C05414=1035.741,-69.357,-80.600,168.332,38.927,157.287
C05415=1035.746,-69.108,-80.612,168.335,38.926,157.287
C05416=1035.752,-68.858,-80.623,168.337,38.926,157.287
C05417=1035.758,-68.609,-80.635,168.340,38.926,157.287
C05418=1035.766,-68.326,-80.648,168.343,38.925,157.287
C05419=1035.773,-68.043,-80.661,168.346,38.925,157.287
C05420=1035.779,-67.760,-80.674,168.349,38.924,157.287
C05421=1035.786,-67.478,-80.687,168.352,38.924,157.287
C05422=1035.793,-67.228,-80.699,168.354,38.923,157.287
C05423=1035.798,-66.978,-80.711,168.357,38.923,157.287
C05424=1035.804,-66.729,-80.723,168.359,38.922,157.287
C05425=1035.811,-66.479,-80.735,168.362,38.922,157.287
C05426=1035.817,-66.229,-80.746,168.365,38.921,157.287
C05427=1035.823,-65.980,-80.758,168.367,38.921,157.287
C05428=1035.829,-65.730,-80.769,168.370,38.921,157.287
C05429=1035.836,-65.480,-80.781,168.371,38.920,157.287
C05430=1035.842,-65.231,-80.793,168.374,38.920,157.287
C05431=1035.847,-64.981,-80.805,168.376,38.919,157.287
C05432=1035.854,-64.731,-80.817,168.379,38.919,157.287
C05433=1035.860,-64.482,-80.828,168.382,38.918,157.287
C05434=1035.866,-64.232,-80.840,168.384,38.918,157.287
C05435=1035.872,-63.982,-80.852,168.387,38.918,157.287
C05436=1035.878,-63.733,-80.864,168.389,38.917,157.287
C05437=1035.885,-63.483,-80.875,168.392,38.917,157.287
C05438=1035.891,-63.234,-80.887,168.394,38.916,157.287
C05439=1035.897,-62.984,-80.899,168.397,38.916,157.287
C05440=1035.903,-62.734,-80.910,168.400,38.915,157.287
C05441=1035.910,-62.485,-80.922,168.402,38.915,157.287
C05442=1035.916,-62.235,-80.934,168.405,38.914,157.287
C05443=1035.921,-61.986,-80.946,168.407,38.914,157.287
C05444=1035.928,-61.736,-80.958,168.410,38.914,157.287
C05445=1035.934,-61.486,-80.970,168.412,38.913,157.287
C05446=1035.940,-61.236,-80.982,168.415,38.913,157.287
C05447=1035.946,-60.987,-80.994,168.418,38.912,157.287
C05448=1035.953,-60.737,-81.005,168.420,38.912,157.287
C05449=1035.959,-60.488,-81.017,168.423,38.911,157.287
C05450=1035.965,-60.238,-81.030,168.425,38.911,157.287
C05451=1035.972,-59.988,-81.042,168.428,38.910,157.287
C05452=1035.978,-59.739,-81.053,168.430,38.910,157.287
C05453=1035.984,-59.489,-81.066,168.433,38.909,157.287
C05454=1035.990,-59.239,-81.077,168.435,38.909,157.287
C05455=1035.997,-58.990,-81.089,168.438,38.908,157.287
C05456=1036.004,-58.740,-81.101,168.441,38.908,157.287
C05457=1036.009,-58.491,-81.113,168.443,38.908,157.287
C05458=1036.015,-58.241,-81.125,168.446,38.907,157.287
C05459=1036.022,-57.992,-81.137,168.448,38.907,157.287
C05460=1036.028,-57.742,-81.150,168.451,38.906,157.287
C05461=1036.034,-57.492,-81.161,168.453,38.906,157.287
C05462=1036.041,-57.242,-81.173,168.456,38.906,157.287
C05463=1036.046,-56.993,-81.185,168.458,38.905,157.287
C05464=1036.053,-56.743,-81.197,168.461,38.905,157.287
C05465=1036.060,-56.494,-81.209,168.464,38.904,157.287
C05466=1036.066,-56.248,-81.221,168.466,38.904,157.287
C05467=1036.072,-56.003,-81.233,168.469,38.904,157.287
C05468=1036.078,-55.758,-81.245,168.470,38.903,157.287
C05469=1036.084,-55.512,-81.257,168.473,38.903,157.287
C05470=1036.090,-55.268,-81.269,168.475,38.902,157.286
C05471=1036.097,-55.022,-81.280,168.478,38.902,157.287
C05472=1036.103,-54.777,-81.293,168.480,38.902,157.287
C05473=1036.109,-54.531,-81.304,168.483,38.901,157.286
C05474=1036.115,-54.282,-81.316,168.485,38.901,157.287
C05475=1036.122,-54.032,-81.328,168.488,38.901,157.287
C05476=1036.128,-53.782,-81.341,168.490,38.900,157.286
C05477=1036.135,-53.533,-81.353,168.493,38.900,157.287
C05478=1036.141,-53.283,-81.365,168.495,38.899,157.286
C05479=1036.147,-53.033,-81.377,168.498,38.899,157.286
C05480=1036.154,-52.784,-81.389,168.500,38.899,157.287
C05481=1036.160,-52.534,-81.401,168.503,38.898,157.286
C05482=1036.168,-52.244,-81.416,168.506,38.898,157.286
C05483=1036.174,-51.954,-81.430,168.509,38.897,157.286
C05484=1036.182,-51.664,-81.444,168.512,38.897,157.286
C05485=1036.190,-51.373,-81.459,168.515,38.896,157.286
C05486=1036.197,-51.124,-81.471,168.517,38.896,157.286
C05487=1036.203,-50.874,-81.483,168.520,38.895,157.286
C05488=1036.209,-50.624,-81.495,168.522,38.895,157.286
C05489=1036.216,-50.375,-81.507,168.525,38.894,157.286
C05490=1036.222,-50.125,-81.520,168.527,38.894,157.286
C05491=1036.228,-49.876,-81.533,168.530,38.894,157.287
C05492=1036.234,-49.626,-81.546,168.532,38.894,157.287
C05493=1036.240,-49.377,-81.557,168.535,38.894,157.287
C05494=1036.246,-49.127,-81.570,168.537,38.893,157.287
C05495=1036.252,-48.878,-81.583,168.539,38.893,157.287
C05496=1036.259,-48.628,-81.595,168.542,38.893,157.287
C05497=1036.265,-48.378,-81.607,168.544,38.893,157.287
C05498=1036.270,-48.129,-81.620,168.547,38.892,157.287
C05499=1036.277,-47.880,-81.633,168.549,38.892,157.287
C05500=1036.283,-47.630,-81.645,168.552,38.892,157.287
C05501=1036.289,-47.380,-81.658,168.554,38.892,157.287
C05502=1036.295,-47.131,-81.671,168.557,38.891,157.287
C05503=1036.302,-46.881,-81.683,168.559,38.891,157.287
C05504=1036.308,-46.631,-81.696,168.562,38.891,157.287
C05505=1036.314,-46.382,-81.709,168.564,38.891,157.287
C05506=1036.320,-46.132,-81.721,168.566,38.891,157.287
C05507=1036.327,-45.882,-81.733,168.569,38.890,157.287
C05508=1036.333,-45.633,-81.747,168.571,38.890,157.287
C05509=1036.339,-45.383,-81.759,168.574,38.889,157.287
C05510=1036.345,-45.134,-81.771,168.576,38.889,157.287
C05511=1036.352,-44.884,-81.785,168.579,38.889,157.287
C05512=1036.358,-44.634,-81.797,168.581,38.889,157.287
C05513=1036.364,-44.385,-81.811,168.584,38.889,157.287
C05514=1036.371,-44.135,-81.823,168.586,38.889,157.287
C05515=1036.377,-43.885,-81.835,168.588,38.889,157.287
C05516=1036.383,-43.636,-81.848,168.591,38.888,157.287
C05517=1036.389,-43.386,-81.861,168.593,38.888,157.287
C05518=1036.396,-43.137,-81.874,168.596,38.887,157.287
C05519=1036.402,-42.887,-81.886,168.598,38.887,157.287
C05520=1036.408,-42.638,-81.899,168.601,38.887,157.287
C05521=1036.414,-42.388,-81.912,168.603,38.887,157.287
C05522=1036.421,-42.139,-81.925,168.606,38.887,157.287
C05523=1036.428,-41.888,-81.938,168.608,38.887,157.287
C05524=1036.434,-41.639,-81.951,168.610,38.887,157.287
C05525=1036.440,-41.389,-81.963,168.613,38.886,157.287
C05526=1036.446,-41.140,-81.977,168.615,38.886,157.287
C05527=1036.453,-40.890,-81.989,168.618,38.885,157.287
C05528=1036.459,-40.641,-82.002,168.620,38.885,157.287
C05529=1036.465,-40.391,-82.014,168.623,38.885,157.287
C05530=1036.471,-40.141,-82.028,168.625,38.885,157.287
C05531=1036.478,-39.892,-82.040,168.627,38.885,157.287
C05532=1036.484,-39.642,-82.053,168.630,38.885,157.288
C05533=1036.490,-39.393,-82.066,168.632,38.885,157.288
C05534=1036.496,-39.143,-82.079,168.635,38.884,157.287
C05535=1036.502,-38.893,-82.092,168.637,38.884,157.288
C05536=1036.510,-38.644,-82.105,168.640,38.883,157.288
C05537=1036.515,-38.394,-82.119,168.642,38.883,157.288
C05538=1036.521,-38.144,-82.131,168.644,38.883,157.288
C05539=1036.528,-37.895,-82.144,168.647,38.883,157.288
C05540=1036.534,-37.646,-82.158,168.649,38.883,157.288
C05541=1036.540,-37.396,-82.170,168.651,38.883,157.288
C05542=1036.546,-37.146,-82.184,168.654,38.883,157.288
C05543=1036.553,-36.897,-82.197,168.656,38.883,157.288
C05544=1036.559,-36.647,-82.210,168.659,38.883,157.288
C05545=1036.565,-36.398,-82.223,168.662,38.883,157.288
C05546=1036.572,-36.117,-82.238,168.665,38.883,157.288
C05547=1036.580,-35.835,-82.253,168.667,38.882,157.288
C05548=1036.586,-35.554,-82.267,168.670,38.882,157.288
C05549=1036.593,-35.273,-82.282,168.673,38.882,157.288
C05550=1036.600,-35.024,-82.296,168.675,38.882,157.288
C05551=1036.606,-34.774,-82.308,168.677,38.882,157.288
C05552=1036.612,-34.524,-82.322,168.680,38.882,157.288
C05553=1036.619,-34.275,-82.335,168.682,38.882,157.288
C05554=1036.625,-34.026,-82.348,168.684,38.881,157.288
C05555=1036.631,-33.776,-82.361,168.687,38.881,157.288
C05556=1036.638,-33.526,-82.375,168.689,38.881,157.288
C05557=1036.644,-33.277,-82.388,168.692,38.881,157.289
C05558=1036.650,-33.027,-82.401,168.694,38.881,157.289
C05559=1036.655,-32.778,-82.415,168.696,38.881,157.289
C05560=1036.662,-32.528,-82.429,168.699,38.880,157.289
C05561=1036.668,-32.278,-82.441,168.701,38.880,157.289
C05562=1036.674,-32.029,-82.454,168.703,38.880,157.289
C05563=1036.681,-31.780,-82.468,168.706,38.880,157.289
C05564=1036.687,-31.530,-82.481,168.708,38.880,157.289
C05565=1036.694,-31.280,-82.495,168.710,38.880,157.289
C05566=1036.700,-31.031,-82.508,168.713,38.880,157.289
C05567=1036.707,-30.781,-82.521,168.715,38.880,157.289
C05568=1036.713,-30.532,-82.535,168.717,38.880,157.289
C05569=1036.719,-30.283,-82.548,168.720,38.880,157.289
C05570=1036.726,-30.032,-82.561,168.722,38.880,157.289
C05571=1036.732,-29.783,-82.574,168.725,38.880,157.289
C05572=1036.738,-29.533,-82.587,168.727,38.879,157.289
C05573=1036.745,-29.283,-82.601,168.729,38.879,157.289
C05574=1036.751,-29.034,-82.614,168.732,38.879,157.289
C05575=1036.757,-28.785,-82.628,168.734,38.879,157.289
C05576=1036.763,-28.535,-82.642,168.736,38.879,157.289
C05577=1036.770,-28.285,-82.655,168.739,38.879,157.289
C05578=1036.776,-28.036,-82.668,168.741,38.879,157.289
C05579=1036.783,-27.786,-82.682,168.743,38.878,157.289
C05580=1036.789,-27.537,-82.695,168.746,38.878,157.289
C05581=1036.796,-27.287,-82.709,168.748,38.878,157.290
C05582=1036.802,-27.038,-82.722,168.750,38.878,157.290
C05583=1036.807,-26.788,-82.736,168.753,38.878,157.290
C05584=1036.814,-26.538,-82.750,168.755,38.878,157.290
C05585=1036.820,-26.289,-82.763,168.757,38.878,157.290
C05586=1036.826,-26.039,-82.777,168.761,38.878,157.290
C05587=1036.833,-25.789,-82.791,168.763,38.878,157.290
C05588=1036.839,-25.541,-82.804,168.765,38.878,157.290
C05589=1036.846,-25.291,-82.818,168.767,38.878,157.290
C05590=1036.851,-25.041,-82.832,168.770,38.878,157.290
C05591=1036.858,-24.792,-82.845,168.772,38.878,157.290
C05592=1036.865,-24.542,-82.859,168.774,38.878,157.290
C05593=1036.870,-24.292,-82.873,168.777,38.878,157.290
C05594=1036.876,-24.043,-82.886,168.779,38.878,157.290
C05595=1036.883,-23.793,-82.901,168.781,38.878,157.290
C05596=1036.889,-23.544,-82.914,168.783,38.878,157.290
C05597=1036.896,-23.294,-82.928,168.786,38.878,157.290
C05598=1036.901,-23.045,-82.942,168.788,38.878,157.290
C05599=1036.908,-22.795,-82.955,168.790,38.878,157.291
C05600=1036.914,-22.546,-82.969,168.793,38.878,157.291
C05601=1036.920,-22.296,-82.983,168.795,38.878,157.291
C05602=1036.927,-22.046,-82.997,168.797,38.878,157.291
C05603=1036.933,-21.797,-83.010,168.799,38.878,157.291
C05604=1036.939,-21.548,-83.025,168.802,38.877,157.291
C05605=1036.946,-21.298,-83.038,168.804,38.878,157.291
C05606=1036.952,-21.048,-83.052,168.806,38.878,157.291
C05607=1036.958,-20.799,-83.066,168.809,38.878,157.291
C05608=1036.965,-20.549,-83.080,168.811,38.878,157.291
C05609=1036.971,-20.300,-83.093,168.813,38.877,157.291
C05610=1036.979,-20.018,-83.110,168.817,38.878,157.291
C05611=1036.985,-19.736,-83.125,168.819,38.878,157.291
C05612=1036.992,-19.454,-83.141,168.822,38.878,157.291
C05613=1036.999,-19.172,-83.157,168.824,38.877,157.291
C05614=1037.006,-18.923,-83.171,168.827,38.877,157.291
C05615=1037.013,-18.673,-83.184,168.829,38.878,157.292
C05616=1037.018,-18.424,-83.198,168.831,38.878,157.292
C05617=1037.025,-18.174,-83.213,168.833,38.878,157.292
C05618=1037.031,-17.925,-83.226,168.836,38.877,157.292
C05619=1037.038,-17.675,-83.240,168.838,38.877,157.292
C05620=1037.044,-17.426,-83.254,168.840,38.877,157.292
C05621=1037.050,-17.176,-83.268,168.843,38.878,157.292
C05622=1037.056,-16.927,-83.282,168.845,38.877,157.292
C05623=1037.063,-16.677,-83.296,168.847,38.877,157.292
C05624=1037.070,-16.427,-83.310,168.849,38.877,157.292
C05625=1037.076,-16.178,-83.324,168.852,38.877,157.292
C05626=1037.082,-15.928,-83.338,168.854,38.878,157.292
C05627=1037.089,-15.680,-83.352,168.856,38.877,157.292
C05628=1037.095,-15.430,-83.366,168.858,38.877,157.292
C05629=1037.101,-15.180,-83.380,168.861,38.877,157.292
C05630=1037.107,-14.930,-83.395,168.863,38.878,157.292
C05631=1037.114,-14.681,-83.408,168.865,38.877,157.293
C05632=1037.120,-14.431,-83.423,168.867,38.877,157.293
C05633=1037.127,-14.182,-83.437,168.870,38.878,157.293
C05634=1037.133,-13.933,-83.451,168.873,38.878,157.293
C05635=1037.139,-13.683,-83.466,168.875,38.878,157.293
C05636=1037.145,-13.434,-83.479,168.877,38.878,157.293
C05637=1037.152,-13.184,-83.494,168.879,38.878,157.293
C05638=1037.157,-12.934,-83.508,168.882,38.878,157.293
C05639=1037.164,-12.685,-83.523,168.884,38.878,157.293
C05640=1037.170,-12.435,-83.537,168.886,38.878,157.293
C05641=1037.176,-12.186,-83.551,168.888,38.878,157.293
C05642=1037.183,-11.936,-83.566,168.890,38.879,157.293
C05643=1037.189,-11.687,-83.580,168.893,38.878,157.293
C05644=1037.196,-11.438,-83.594,168.895,38.878,157.293
C05645=1037.202,-11.188,-83.609,168.897,38.878,157.293
C05646=1037.208,-10.938,-83.623,168.899,38.879,157.294
C05647=1037.215,-10.689,-83.637,168.901,38.879,157.294
C05648=1037.221,-10.439,-83.651,168.904,38.878,157.294
C05649=1037.227,-10.190,-83.666,168.906,38.879,157.294
C05650=1037.234,-9.940,-83.680,168.908,38.879,157.294
C05651=1037.239,-9.691,-83.694,168.910,38.879,157.294
C05652=1037.246,-9.441,-83.709,168.913,38.879,157.294
C05653=1037.253,-9.192,-83.723,168.916,38.879,157.294
C05654=1037.258,-8.943,-83.738,168.918,38.879,157.294
C05655=1037.264,-8.693,-83.752,168.920,38.879,157.294
C05656=1037.272,-8.443,-83.767,168.922,38.879,157.294
C05657=1037.277,-8.194,-83.781,168.924,38.879,157.294
C05658=1037.283,-7.944,-83.795,168.927,38.880,157.295
C05659=1037.291,-7.695,-83.810,168.929,38.880,157.295
C05660=1037.297,-7.445,-83.825,168.931,38.879,157.295
C05661=1037.303,-7.196,-83.839,168.933,38.880,157.295
C05662=1037.310,-6.946,-83.853,168.935,38.880,157.295
C05663=1037.316,-6.696,-83.868,168.938,38.880,157.295
C05664=1037.322,-6.447,-83.882,168.940,38.880,157.295
C05665=1037.328,-6.198,-83.897,168.942,38.880,157.295
C05666=1037.335,-5.948,-83.911,168.944,38.880,157.295
C05667=1037.341,-5.698,-83.926,168.946,38.880,157.295
C05668=1037.347,-5.449,-83.941,168.949,38.880,157.295
C05669=1037.354,-5.200,-83.955,168.951,38.880,157.295
C05670=1037.361,-4.950,-83.970,168.953,38.880,157.295
C05671=1037.367,-4.701,-83.985,168.956,38.881,157.295
C05672=1037.373,-4.451,-83.998,168.958,38.880,157.296
C05673=1037.380,-4.202,-84.013,168.960,38.880,157.296
C05674=1037.387,-3.918,-84.029,168.963,38.881,157.296
C05675=1037.394,-3.635,-84.046,168.965,38.881,157.296
C05676=1037.402,-3.351,-84.063,168.968,38.881,157.296
C05677=1037.408,-3.067,-84.080,168.970,38.881,157.296
C05678=1037.414,-2.818,-84.095,168.972,38.881,157.296
C05679=1037.420,-2.569,-84.110,168.975,38.881,157.296
C05680=1037.427,-2.319,-84.125,168.977,38.882,157.296
C05681=1037.433,-2.069,-84.139,168.979,38.882,157.296
C05682=1037.439,-1.820,-84.154,168.981,38.882,157.296
C05683=1037.445,-1.571,-84.169,168.983,38.882,157.297
C05684=1037.452,-1.321,-84.184,168.985,38.883,157.297
C05685=1037.458,-1.071,-84.199,168.987,38.882,157.297
C05686=1037.464,-0.823,-84.213,168.990,38.883,157.297
C05687=1037.470,-0.573,-84.228,168.993,38.883,157.297
C05688=1037.476,-0.323,-84.243,168.995,38.883,157.297
C05689=1037.483,-0.074,-84.258,168.997,38.883,157.297
C05690=1037.489,0.175,-84.273,168.999,38.884,157.297
C05691=1037.495,0.425,-84.288,169.001,38.884,157.297
C05692=1037.501,0.675,-84.303,169.003,38.884,157.297
C05693=1037.508,0.924,-84.318,169.005,38.884,157.297
C05694=1037.514,1.173,-84.333,169.007,38.885,157.298
C05695=1037.520,1.422,-84.348,169.009,38.884,157.298
C05696=1037.527,1.672,-84.363,169.012,38.884,157.298
C05697=1037.533,1.922,-84.378,169.014,38.885,157.298
C05698=1037.539,2.171,-84.393,169.016,38.885,157.298
C05699=1037.546,2.421,-84.408,169.019,38.885,157.298
C05700=1037.552,2.671,-84.423,169.021,38.885,157.298
C05701=1037.558,2.920,-84.437,169.023,38.886,157.298
C05702=1037.565,3.169,-84.453,169.025,38.885,157.298
C05703=1037.571,3.418,-84.468,169.027,38.886,157.298
C05704=1037.577,3.668,-84.483,169.029,38.886,157.298
C05705=1037.584,3.918,-84.498,169.032,38.886,157.299
C05706=1037.590,4.167,-84.513,169.034,38.886,157.299
C05707=1037.595,4.417,-84.528,169.036,38.887,157.299
C05708=1037.602,4.666,-84.544,169.038,38.887,157.299
C05709=1037.608,4.915,-84.559,169.040,38.887,157.299
C05710=1037.615,5.165,-84.573,169.042,38.887,157.299
C05711=1037.621,5.415,-84.588,169.044,38.888,157.299
C05712=1037.627,5.664,-84.603,169.046,38.887,157.299
C05713=1037.634,5.913,-84.619,169.049,38.888,157.299
C05714=1037.641,6.163,-84.634,169.052,38.888,157.299
C05715=1037.647,6.413,-84.649,169.054,38.888,157.299
C05716=1037.653,6.662,-84.663,169.056,38.888,157.300
C05717=1037.659,6.911,-84.679,169.058,38.888,157.300
C05718=1037.666,7.160,-84.694,169.060,38.889,157.300
C05719=1037.672,7.410,-84.709,169.062,38.888,157.300
C05720=1037.679,7.660,-84.724,169.064,38.889,157.300
C05721=1037.685,7.909,-84.740,169.066,38.889,157.300
C05722=1037.691,8.159,-84.755,169.068,38.889,157.300
C05723=1037.697,8.408,-84.770,169.070,38.889,157.300
C05724=1037.704,8.657,-84.786,169.073,38.890,157.300
C05725=1037.710,8.907,-84.801,169.075,38.890,157.300
C05726=1037.717,9.157,-84.816,169.077,38.889,157.300
C05727=1037.723,9.406,-84.831,169.080,38.890,157.301
C05728=1037.730,9.655,-84.846,169.082,38.890,157.301
C05729=1037.736,9.905,-84.861,169.084,38.890,157.301
C05730=1037.743,10.154,-84.877,169.086,38.890,157.301
C05731=1037.749,10.404,-84.892,169.088,38.891,157.301
C05732=1037.756,10.653,-84.907,169.090,38.891,157.301
C05733=1037.762,10.902,-84.922,169.092,38.891,157.301
C05734=1037.768,11.152,-84.938,169.095,38.891,157.301
C05735=1037.774,11.402,-84.953,169.097,38.891,157.301
C05736=1037.781,11.651,-84.969,169.099,38.891,157.301
C05737=1037.787,11.901,-84.984,169.101,38.891,157.301
C05738=1037.795,12.186,-85.001,169.103,38.892,157.301
C05739=1037.802,12.471,-85.019,169.106,38.892,157.302
C05740=1037.810,12.757,-85.036,169.108,38.892,157.302
C05741=1037.817,13.042,-85.054,169.110,38.892,157.302
C05742=1037.824,13.291,-85.069,169.114,38.892,157.302
C05743=1037.830,13.541,-85.084,169.116,38.892,157.302
C05744=1037.836,13.790,-85.100,169.118,38.893,157.302
C05745=1037.843,14.040,-85.115,169.120,38.893,157.302
C05746=1037.849,14.289,-85.131,169.122,38.893,157.302
C05747=1037.856,14.538,-85.146,169.124,38.893,157.302
C05748=1037.862,14.788,-85.162,169.126,38.894,157.302
C05749=1037.868,15.037,-85.177,169.128,38.893,157.302
C05750=1037.875,15.287,-85.193,169.130,38.894,157.303
C05751=1037.880,15.536,-85.208,169.132,38.895,157.303
C05752=1037.887,15.786,-85.224,169.134,38.894,157.303
C05753=1037.893,16.035,-85.240,169.136,38.895,157.303
C05754=1037.899,16.285,-85.255,169.138,38.895,157.303
C05755=1037.906,16.534,-85.271,169.141,38.895,157.303
C05756=1037.912,16.784,-85.286,169.143,38.895,157.303
C05757=1037.918,17.033,-85.302,169.145,38.896,157.303
C05758=1037.925,17.282,-85.318,169.147,38.896,157.303
C05759=1037.931,17.532,-85.333,169.149,38.896,157.304
C05760=1037.937,17.781,-85.349,169.151,38.897,157.304
C05761=1037.943,18.030,-85.365,169.153,38.896,157.304
C05762=1037.950,18.280,-85.381,169.156,38.897,157.304
C05763=1037.957,18.529,-85.396,169.158,38.897,157.304
C05764=1037.963,18.779,-85.412,169.160,38.897,157.304
C05765=1037.969,19.028,-85.427,169.162,38.897,157.304
C05766=1037.976,19.277,-85.443,169.164,38.898,157.304
C05767=1037.982,19.527,-85.459,169.167,38.898,157.304
C05768=1037.988,19.776,-85.474,169.169,38.898,157.304
C05769=1037.994,20.026,-85.491,169.171,38.899,157.305
C05770=1038.001,20.275,-85.506,169.173,38.899,157.305
C05771=1038.007,20.525,-85.522,169.175,38.899,157.305
C05772=1038.014,20.775,-85.538,169.177,38.900,157.305
C05773=1038.020,21.024,-85.554,169.179,38.899,157.305
C05774=1038.027,21.273,-85.570,169.181,38.900,157.305
C05775=1038.033,21.522,-85.586,169.183,38.900,157.305
C05776=1038.039,21.772,-85.601,169.185,38.900,157.305
C05777=1038.045,22.021,-85.617,169.187,38.901,157.305
C05778=1038.052,22.270,-85.633,169.189,38.901,157.305
C05779=1038.058,22.520,-85.649,169.192,38.901,157.306
C05780=1038.065,22.769,-85.665,169.194,38.902,157.306
C05781=1038.071,23.019,-85.681,169.196,38.902,157.306
C05782=1038.077,23.268,-85.696,169.198,38.902,157.306
C05783=1038.083,23.518,-85.713,169.200,38.902,157.306
C05784=1038.090,23.767,-85.728,169.202,38.903,157.306
C05785=1038.096,24.016,-85.744,169.204,38.903,157.306
C05786=1038.102,24.265,-85.761,169.206,38.903,157.306
C05787=1038.109,24.516,-85.776,169.208,38.904,157.306
C05788=1038.115,24.765,-85.792,169.210,38.903,157.307
C05789=1038.121,25.014,-85.808,169.212,38.904,157.307
C05790=1038.127,25.264,-85.824,169.215,38.904,157.307
C05791=1038.134,25.513,-85.840,169.217,38.904,157.307
C05792=1038.141,25.763,-85.856,169.219,38.905,157.307
C05793=1038.147,26.012,-85.872,169.221,38.905,157.307
C05794=1038.153,26.261,-85.888,169.223,38.905,157.307
C05795=1038.159,26.510,-85.905,169.225,38.906,157.307
C05796=1038.166,26.759,-85.920,169.227,38.906,157.307
C05797=1038.172,27.009,-85.937,169.229,38.906,157.308
C05798=1038.179,27.258,-85.953,169.231,38.906,157.308
C05799=1038.185,27.508,-85.969,169.233,38.907,157.308
C05800=1038.191,27.758,-85.984,169.235,38.907,157.308
C05801=1038.198,28.008,-86.000,169.237,38.907,157.308
C05802=1038.205,28.294,-86.019,169.240,38.907,157.308
C05803=1038.212,28.580,-86.038,169.243,38.908,157.308
C05804=1038.219,28.867,-86.056,169.245,38.908,157.308
C05805=1038.226,29.153,-86.075,169.247,38.908,157.308
C05806=1038.233,29.404,-86.092,169.249,38.909,157.309
C05807=1038.239,29.653,-86.108,169.251,38.909,157.309
C05808=1038.246,29.902,-86.123,169.253,38.910,157.309
C05809=1038.252,30.151,-86.140,169.255,38.910,157.309
C05810=1038.258,30.401,-86.156,169.257,38.910,157.309
C05811=1038.264,30.650,-86.173,169.260,38.911,157.309
C05812=1038.271,30.899,-86.189,169.262,38.911,157.309
C05813=1038.277,31.148,-86.205,169.264,38.911,157.309
C05814=1038.284,31.398,-86.222,169.266,38.912,157.310
C05815=1038.290,31.648,-86.238,169.268,38.912,157.310
C05816=1038.296,31.897,-86.254,169.270,38.912,157.310
C05817=1038.302,32.146,-86.270,169.272,38.913,157.310
C05818=1038.309,32.396,-86.287,169.274,38.912,157.310
C05819=1038.315,32.645,-86.304,169.276,38.913,157.310
C05820=1038.321,32.894,-86.320,169.278,38.913,157.310
C05821=1038.327,33.144,-86.336,169.280,38.913,157.310
C05822=1038.334,33.393,-86.352,169.283,38.914,157.310
C05823=1038.340,33.643,-86.368,169.285,38.914,157.311
C05824=1038.346,33.891,-86.385,169.287,38.915,157.311
C05825=1038.353,34.142,-86.402,169.289,38.915,157.311
C05826=1038.360,34.391,-86.418,169.291,38.915,157.311
C05827=1038.366,34.640,-86.434,169.293,38.916,157.311
C05828=1038.372,34.890,-86.451,169.295,38.916,157.311
C05829=1038.378,35.139,-86.467,169.297,38.916,157.311
C05830=1038.384,35.388,-86.484,169.299,38.917,157.311
C05831=1038.392,35.638,-86.500,169.301,38.917,157.311
C05832=1038.398,35.887,-86.516,169.303,38.917,157.312
C05833=1038.404,36.136,-86.533,169.305,38.917,157.312
C05834=1038.410,36.386,-86.550,169.307,38.918,157.312
C05835=1038.416,36.635,-86.566,169.309,38.918,157.312
C05836=1038.422,36.885,-86.582,169.311,38.918,157.312
C05837=1038.430,37.134,-86.599,169.313,38.918,157.312
C05838=1038.436,37.383,-86.615,169.315,38.919,157.312
C05839=1038.442,37.633,-86.632,169.317,38.920,157.312
C05840=1038.449,37.882,-86.649,169.319,38.919,157.312
C05841=1038.455,38.131,-86.665,169.321,38.920,157.313
C05842=1038.461,38.381,-86.682,169.323,38.920,157.313
C05843=1038.467,38.630,-86.699,169.326,38.921,157.313
C05844=1038.473,38.879,-86.715,169.328,38.921,157.313
C05845=1038.480,39.129,-86.732,169.330,38.921,157.313
C05846=1038.486,39.378,-86.748,169.332,38.922,157.313
C05847=1038.492,39.627,-86.765,169.334,38.922,157.313
C05848=1038.499,39.877,-86.782,169.336,38.922,157.313
C05849=1038.505,40.126,-86.798,169.338,38.923,157.314
C05850=1038.512,40.376,-86.816,169.340,38.923,157.314
C05851=1038.517,40.625,-86.832,169.342,38.924,157.314
C05852=1038.523,40.874,-86.849,169.344,38.924,157.314
C05853=1038.530,41.124,-86.866,169.346,38.924,157.314
C05854=1038.536,41.373,-86.882,169.348,38.925,157.314
C05855=1038.543,41.623,-86.900,169.350,38.925,157.314
C05856=1038.549,41.872,-86.916,169.352,38.926,157.315
C05857=1038.555,42.121,-86.933,169.354,38.926,157.315
C05858=1038.561,42.371,-86.950,169.356,38.926,157.315
C05859=1038.568,42.620,-86.966,169.358,38.927,157.315
C05860=1038.574,42.870,-86.983,169.360,38.927,157.315
C05861=1038.581,43.119,-87.000,169.362,38.927,157.315
C05862=1038.586,43.368,-87.016,169.365,38.928,157.315
C05863=1038.593,43.617,-87.034,169.367,38.928,157.315
C05864=1038.599,43.866,-87.051,169.369,38.929,157.315
C05865=1038.605,44.116,-87.068,169.370,38.929,157.316
C05866=1038.612,44.403,-87.087,169.373,38.930,157.316
C05867=1038.619,44.689,-87.107,169.375,38.930,157.316
C05868=1038.626,44.976,-87.127,169.377,38.931,157.316
C05869=1038.634,45.262,-87.146,169.379,38.931,157.316
C05870=1038.640,45.512,-87.163,169.382,38.932,157.316
C05871=1038.646,45.761,-87.180,169.384,38.932,157.317
C05872=1038.653,46.010,-87.198,169.386,38.932,157.317
C05873=1038.658,46.260,-87.214,169.388,38.933,157.317
C05874=1038.664,46.509,-87.231,169.390,38.933,157.317
C05875=1038.671,46.758,-87.249,169.392,38.934,157.317
C05876=1038.676,47.008,-87.266,169.394,38.934,157.317
C05877=1038.683,47.257,-87.283,169.395,38.935,157.317
C05878=1038.690,47.506,-87.300,169.398,38.935,157.318
C05879=1038.695,47.756,-87.317,169.400,38.935,157.318
C05880=1038.702,48.005,-87.334,169.402,38.936,157.318
C05881=1038.708,48.254,-87.351,169.404,38.936,157.318
C05882=1038.715,48.503,-87.368,169.406,38.937,157.318
C05883=1038.721,48.754,-87.386,169.408,38.937,157.318
C05884=1038.727,49.002,-87.403,169.410,38.938,157.318
C05885=1038.734,49.252,-87.420,169.412,38.938,157.318
C05886=1038.739,49.501,-87.437,169.414,38.938,157.319
C05887=1038.746,49.751,-87.454,169.416,38.939,157.319
C05888=1038.752,50.000,-87.471,169.418,38.939,157.319
C05889=1038.758,50.249,-87.489,169.420,38.940,157.319
C05890=1038.764,50.498,-87.506,169.422,38.940,157.319
C05891=1038.771,50.748,-87.523,169.424,38.941,157.319
C05892=1038.776,50.997,-87.540,169.426,38.941,157.319
C05893=1038.783,51.247,-87.557,169.428,38.941,157.319
C05894=1038.790,51.495,-87.574,169.430,38.942,157.320
C05895=1038.796,51.745,-87.592,169.432,38.942,157.320
C05896=1038.802,51.994,-87.609,169.435,38.943,157.320
C05897=1038.808,52.244,-87.626,169.436,38.943,157.320
C05898=1038.814,52.493,-87.644,169.438,38.943,157.320
C05899=1038.821,52.742,-87.661,169.440,38.944,157.320
C05900=1038.828,52.992,-87.678,169.442,38.944,157.320
C05901=1038.833,53.241,-87.696,169.444,38.945,157.321
C05902=1038.840,53.490,-87.713,169.446,38.945,157.321
C05903=1038.845,53.740,-87.730,169.448,38.945,157.321
C05904=1038.852,53.989,-87.747,169.450,38.946,157.321
C05905=1038.858,54.238,-87.764,169.453,38.946,157.321
C05906=1038.865,54.488,-87.782,169.455,38.947,157.321
C05907=1038.871,54.737,-87.800,169.457,38.947,157.321
C05908=1038.878,54.986,-87.817,169.458,38.947,157.321
C05909=1038.884,55.236,-87.834,169.460,38.948,157.322
C05910=1038.890,55.484,-87.851,169.462,38.948,157.322
C05911=1038.897,55.734,-87.869,169.464,38.949,157.322
C05912=1038.903,55.984,-87.887,169.466,38.949,157.322
C05913=1038.909,56.232,-87.904,169.468,38.949,157.322
C05914=1038.916,56.482,-87.921,169.471,38.949,157.322
C05915=1038.922,56.731,-87.939,169.473,38.950,157.322
C05916=1038.929,56.980,-87.956,169.475,38.950,157.322
C05917=1038.934,57.231,-87.973,169.477,38.951,157.323
C05918=1038.941,57.479,-87.990,169.479,38.951,157.323
C05919=1038.947,57.729,-88.007,169.480,38.951,157.323
C05920=1038.954,57.978,-88.025,169.482,38.952,157.323
C05921=1038.960,58.227,-88.042,169.484,38.952,157.323
C05922=1038.967,58.477,-88.060,169.486,38.952,157.323
C05923=1038.973,58.726,-88.078,169.488,38.953,157.323
C05924=1038.979,58.974,-88.095,169.491,38.953,157.323
C05925=1038.985,59.224,-88.113,169.493,38.954,157.324
C05926=1038.992,59.474,-88.131,169.495,38.954,157.324
C05927=1038.999,59.723,-88.148,169.497,38.954,157.324
C05928=1039.005,59.972,-88.166,169.499,38.955,157.324
C05929=1039.012,60.221,-88.183,169.501,38.955,157.324
C05930=1039.019,60.507,-88.203,169.503,38.956,157.324
C05931=1039.026,60.794,-88.223,169.505,38.956,157.324
C05932=1039.034,61.081,-88.243,169.507,38.956,157.324
C05933=1039.041,61.367,-88.263,169.510,38.957,157.325
C05934=1039.047,61.616,-88.281,169.512,38.957,157.325
C05935=1039.054,61.866,-88.299,169.514,38.958,157.325
C05936=1039.060,62.115,-88.316,169.516,38.958,157.325
C05937=1039.067,62.364,-88.333,169.518,38.958,157.325
C05938=1039.073,62.613,-88.352,169.520,38.959,157.325
C05939=1039.080,62.863,-88.369,169.522,38.959,157.325
C05940=1039.086,63.112,-88.387,169.524,38.959,157.325
C05941=1039.092,63.361,-88.404,169.526,38.959,157.326
C05942=1039.099,63.610,-88.421,169.529,38.960,157.326
C05943=1039.105,63.860,-88.439,169.531,38.961,157.326
C05944=1039.111,64.109,-88.457,169.533,38.961,157.326
C05945=1039.118,64.358,-88.475,169.534,38.961,157.326
C05946=1039.124,64.608,-88.493,169.536,38.961,157.326
C05947=1039.130,64.857,-88.511,169.538,38.962,157.326
C05948=1039.137,65.106,-88.528,169.540,38.963,157.327
C05949=1039.143,65.355,-88.546,169.542,38.963,157.327
C05950=1039.149,65.605,-88.564,169.544,38.964,157.327
C05951=1039.155,65.854,-88.581,169.547,38.964,157.327
C05952=1039.162,66.103,-88.600,169.549,38.965,157.327
C05953=1039.168,66.353,-88.618,169.551,38.965,157.327
C05954=1039.175,66.602,-88.635,169.552,38.965,157.327
C05955=1039.181,66.851,-88.654,169.554,38.965,157.328
C05956=1039.187,67.100,-88.671,169.556,38.966,157.328
C05957=1039.194,67.350,-88.689,169.558,38.967,157.328
C05958=1039.200,67.599,-88.707,169.560,38.967,157.328
C05959=1039.206,67.849,-88.725,169.563,38.968,157.328
C05960=1039.212,68.098,-88.743,169.565,38.968,157.328
C05961=1039.219,68.346,-88.761,169.567,38.969,157.328
C05962=1039.225,68.596,-88.779,169.568,38.968,157.328
C05963=1039.231,68.845,-88.797,169.570,38.969,157.329
C05964=1039.237,69.095,-88.815,169.572,38.970,157.329
C05965=1039.244,69.344,-88.832,169.574,38.970,157.329
C05966=1039.250,69.593,-88.851,169.576,38.971,157.329
C05967=1039.256,69.843,-88.869,169.579,38.971,157.329
C05968=1039.263,70.092,-88.888,169.581,38.972,157.329
C05969=1039.268,70.341,-88.905,169.583,38.972,157.330
C05970=1039.275,70.590,-88.924,169.584,38.973,157.330
C05971=1039.281,70.839,-88.941,169.586,38.973,157.330
C05972=1039.288,71.088,-88.960,169.588,38.974,157.330
C05973=1039.294,71.338,-88.978,169.590,38.974,157.330
C05974=1039.300,71.587,-88.995,169.592,38.975,157.330
C05975=1039.306,71.836,-89.014,169.595,38.975,157.330
C05976=1039.312,72.085,-89.033,169.597,38.975,157.330
C05977=1039.319,72.335,-89.050,169.599,38.976,157.331
C05978=1039.325,72.584,-89.069,169.600,38.976,157.331
C05979=1039.332,72.834,-89.086,169.602,38.977,157.331
C05980=1039.338,73.082,-89.105,169.604,38.977,157.331
C05981=1039.344,73.332,-89.123,169.606,38.978,157.331
C05982=1039.350,73.581,-89.141,169.608,38.978,157.331
C05983=1039.356,73.831,-89.159,169.611,38.979,157.332
C05984=1039.363,74.080,-89.178,169.613,38.979,157.332
C05985=1039.369,74.330,-89.196,169.615,38.980,157.332
C05986=1039.375,74.578,-89.214,169.616,38.980,157.332
C05987=1039.381,74.827,-89.233,169.618,38.981,157.332
C05988=1039.387,75.077,-89.251,169.620,38.981,157.332
C05989=1039.394,75.326,-89.269,169.622,38.982,157.332
C05990=1039.400,75.576,-89.287,169.624,38.982,157.333
C05991=1039.407,75.825,-89.305,169.626,38.982,157.333
C05992=1039.413,76.074,-89.324,169.629,38.983,157.333
C05993=1039.419,76.323,-89.342,169.631,38.983,157.333
C05994=1039.426,76.609,-89.363,169.633,38.984,157.333
C05995=1039.434,76.895,-89.384,169.635,38.984,157.333
C05996=1039.441,77.181,-89.406,169.637,38.985,157.333
C05997=1039.448,77.467,-89.427,169.639,38.985,157.334
C05998=1039.454,77.716,-89.444,169.641,38.986,157.334
C05999=1039.461,77.966,-89.463,169.644,38.986,157.334
C06000=1039.467,78.215,-89.482,169.646,38.987,157.334
C06001=1039.473,78.465,-89.500,169.648,38.987,157.334
C06002=1039.479,78.714,-89.519,169.650,38.988,157.334
C06003=1039.485,78.963,-89.538,169.651,38.988,157.335
C06004=1039.492,79.212,-89.556,169.653,38.989,157.335
C06005=1039.498,79.461,-89.574,169.655,38.990,157.335
C06006=1039.504,79.710,-89.592,169.658,38.990,157.335
C06007=1039.510,79.960,-89.612,169.660,38.991,157.335
C06008=1039.516,80.209,-89.630,169.662,38.992,157.335
C06009=1039.522,80.458,-89.649,169.664,38.992,157.336
C06010=1039.529,80.707,-89.668,169.665,38.993,157.336
C06011=1039.535,80.957,-89.686,169.667,38.993,157.336
C06012=1039.541,81.206,-89.704,169.669,38.994,157.336
C06013=1039.547,81.455,-89.723,169.672,38.994,157.336
C06014=1039.553,81.705,-89.742,169.674,38.995,157.336
C06015=1039.560,81.954,-89.761,169.676,38.995,157.337
C06016=1039.566,82.203,-89.779,169.678,38.996,157.337
C06017=1039.573,82.452,-89.798,169.679,38.996,157.337
C06018=1039.578,82.701,-89.816,169.681,38.997,157.337
C06019=1039.584,82.950,-89.835,169.683,38.997,157.337
C06020=1039.590,83.199,-89.854,169.686,38.998,157.337
C06021=1039.597,83.449,-89.872,169.688,38.998,157.337
C06022=1039.603,83.698,-89.891,169.690,38.999,157.338
C06023=1039.609,83.947,-89.910,169.692,38.999,157.338
C06024=1039.615,84.196,-89.929,169.694,39.000,157.338
C06025=1039.622,84.445,-89.947,169.695,39.000,157.338
C06026=1039.628,84.695,-89.966,169.697,39.001,157.338
C06027=1039.635,84.944,-89.985,169.699,39.001,157.338
C06028=1039.640,85.193,-90.004,169.702,39.002,157.339
C06029=1039.647,85.442,-90.023,169.704,39.002,157.339
C06030=1039.653,85.691,-90.041,169.706,39.003,157.339
C06031=1039.660,85.940,-90.060,169.708,39.003,157.339
C06032=1039.666,86.190,-90.078,169.710,39.004,157.339
C06033=1039.671,86.440,-90.097,169.711,39.004,157.339
C06034=1039.678,86.689,-90.116,169.713,39.005,157.339
C06035=1039.685,86.937,-90.135,169.716,39.005,157.340
C06036=1039.692,87.187,-90.154,169.718,39.005,157.340
C06037=1039.697,87.436,-90.173,169.720,39.006,157.340
C06038=1039.704,87.686,-90.192,169.722,39.006,157.340
C06039=1039.710,87.935,-90.211,169.724,39.007,157.340
C06040=1039.717,88.184,-90.229,169.726,39.007,157.340
C06041=1039.723,88.433,-90.248,169.728,39.008,157.340
C06042=1039.729,88.682,-90.267,169.729,39.008,157.341
C06043=1039.735,88.932,-90.286,169.731,39.009,157.341
C06044=1039.742,89.181,-90.304,169.734,39.009,157.341
C06045=1039.748,89.430,-90.323,169.736,39.010,157.341
C06046=1039.754,89.679,-90.342,169.738,39.010,157.341
C06047=1039.760,89.928,-90.361,169.740,39.011,157.341
C06048=1039.766,90.177,-90.380,169.742,39.011,157.341
C06049=1039.772,90.427,-90.399,169.744,39.012,157.342
C06050=1039.779,90.675,-90.418,169.746,39.012,157.342
C06051=1039.785,90.926,-90.438,169.748,39.013,157.342
C06052=1039.792,91.175,-90.456,169.750,39.014,157.342
C06053=1039.797,91.424,-90.476,169.752,39.015,157.342
C06054=1039.804,91.673,-90.494,169.754,39.015,157.343
C06055=1039.810,91.922,-90.514,169.756,39.016,157.343
C06056=1039.816,92.171,-90.533,169.758,39.016,157.343
C06057=1039.822,92.421,-90.552,169.760,39.017,157.343
C06058=1039.829,92.707,-90.574,169.763,39.017,157.343
C06059=1039.836,92.993,-90.596,169.765,39.018,157.343
C06060=1039.844,93.279,-90.618,169.767,39.019,157.344
C06061=1039.850,93.564,-90.640,169.769,39.019,157.344
C06062=1039.857,93.814,-90.659,169.771,39.020,157.344
C06063=1039.863,94.063,-90.678,169.773,39.020,157.344
C06064=1039.869,94.312,-90.698,169.776,39.021,157.344
C06065=1039.876,94.561,-90.717,169.778,39.021,157.344
C06066=1039.881,94.811,-90.736,169.780,39.022,157.345
C06067=1039.888,95.059,-90.755,169.781,39.022,157.345
C06068=1039.894,95.308,-90.775,169.783,39.023,157.345
C06069=1039.900,95.558,-90.793,169.785,39.023,157.345
C06070=1039.907,95.807,-90.813,169.787,39.024,157.345
C06071=1039.913,96.056,-90.832,169.790,39.025,157.345
C06072=1039.919,96.306,-90.851,169.792,39.026,157.346
C06073=1039.925,96.554,-90.871,169.794,39.026,157.346
C06074=1039.931,96.804,-90.890,169.796,39.027,157.346
C06075=1039.937,97.053,-90.909,169.797,39.027,157.346
C06076=1039.944,97.302,-90.929,169.799,39.028,157.346
C06077=1039.950,97.552,-90.948,169.801,39.028,157.346
C06078=1039.956,97.801,-90.967,169.804,39.029,157.347
C06079=1039.962,98.050,-90.987,169.806,39.029,157.347
C06080=1039.969,98.299,-91.005,169.808,39.030,157.347
C06081=1039.975,98.548,-91.025,169.810,39.030,157.347
C06082=1039.982,98.797,-91.044,169.812,39.031,157.347
C06083=1039.987,99.047,-91.064,169.814,39.031,157.347
C06084=1039.994,99.295,-91.083,169.816,39.032,157.347
C06085=1040.000,99.545,-91.102,169.818,39.032,157.348
C06086=1040.007,99.793,-91.122,169.820,39.033,157.348
C06087=1040.013,100.043,-91.141,169.822,39.033,157.348
C06088=1040.019,100.292,-91.161,169.824,39.034,157.348
C06089=1040.025,100.541,-91.180,169.826,39.034,157.348
C06090=1040.031,100.790,-91.200,169.828,39.035,157.349
C06091=1040.037,101.040,-91.219,169.830,39.036,157.349
C06092=1040.044,101.289,-91.239,169.833,39.036,157.349
C06093=1040.050,101.538,-91.258,169.834,39.037,157.349
C06094=1040.056,101.787,-91.278,169.836,39.037,157.349
C06095=1040.062,102.036,-91.298,169.838,39.038,157.349
C06096=1040.068,102.285,-91.317,169.840,39.039,157.350
C06097=1040.074,102.535,-91.338,169.842,39.040,157.350
C06098=1040.081,102.784,-91.356,169.845,39.040,157.350
C06099=1040.087,103.033,-91.376,169.847,39.041,157.350
C06100=1040.092,103.282,-91.395,169.849,39.041,157.350
C06101=1040.099,103.532,-91.416,169.851,39.042,157.350
C06102=1040.105,103.780,-91.436,169.852,39.043,157.351
C06103=1040.111,104.030,-91.455,169.854,39.043,157.351
C06104=1040.117,104.278,-91.474,169.856,39.044,157.351
C06105=1040.123,104.527,-91.494,169.859,39.044,157.351
C06106=1040.130,104.777,-91.514,169.861,39.045,157.351
C06107=1040.136,105.026,-91.534,169.863,39.045,157.351
C06108=1040.142,105.275,-91.554,169.865,39.046,157.352
C06109=1040.149,105.525,-91.573,169.867,39.047,157.352
C06110=1040.155,105.774,-91.593,169.869,39.047,157.352
C06111=1040.161,106.022,-91.613,169.871,39.048,157.352
C06112=1040.166,106.272,-91.632,169.873,39.048,157.352
C06113=1040.173,106.521,-91.652,169.875,39.049,157.352
C06114=1040.179,106.770,-91.672,169.877,39.049,157.353
C06115=1040.186,107.019,-91.692,169.879,39.050,157.353
C06116=1040.192,107.269,-91.711,169.881,39.050,157.353
C06117=1040.198,107.518,-91.731,169.883,39.052,157.353
C06118=1040.204,107.766,-91.751,169.886,39.052,157.353
C06119=1040.210,108.015,-91.771,169.888,39.053,157.354
C06120=1040.216,108.265,-91.791,169.890,39.053,157.354
C06121=1040.223,108.514,-91.810,169.892,39.054,157.354
C06122=1040.230,108.800,-91.833,169.894,39.054,157.354
C06123=1040.237,109.086,-91.855,169.896,39.055,157.354
C06124=1040.244,109.372,-91.879,169.899,39.056,157.354
C06125=1040.251,109.658,-91.902,169.901,39.056,157.355
C06126=1040.258,109.907,-91.921,169.903,39.057,157.355
C06127=1040.264,110.156,-91.941,169.905,39.057,157.355
C06128=1040.270,110.405,-91.961,169.907,39.058,157.355
C06129=1040.276,110.654,-91.981,169.909,39.059,157.355
C06130=1040.283,110.904,-92.001,169.912,39.059,157.356
C06131=1040.289,111.153,-92.021,169.914,39.060,157.356
C06132=1040.295,111.402,-92.041,169.916,39.060,157.356
C06133=1040.301,111.651,-92.061,169.918,39.061,157.356
C06134=1040.307,111.900,-92.081,169.920,39.062,157.356
C06135=1040.313,112.149,-92.101,169.921,39.063,157.356
C06136=1040.320,112.398,-92.121,169.923,39.063,157.357
C06137=1040.326,112.647,-92.141,169.926,39.064,157.357
C06138=1040.332,112.896,-92.161,169.928,39.064,157.357
C06139=1040.338,113.146,-92.182,169.930,39.065,157.357
C06140=1040.344,113.394,-92.201,169.932,39.066,157.357
C06141=1040.351,113.644,-92.222,169.934,39.066,157.357
C06142=1040.357,113.893,-92.242,169.936,39.067,157.358
C06143=1040.362,114.142,-92.262,169.939,39.068,157.358
C06144=1040.369,114.391,-92.283,169.941,39.068,157.358
C06145=1040.375,114.640,-92.303,169.943,39.069,157.358
C06146=1040.381,114.889,-92.323,169.944,39.070,157.359
C06147=1040.387,115.139,-92.343,169.946,39.071,157.359
C06148=1040.393,115.388,-92.363,169.948,39.071,157.359
C06149=1040.399,115.636,-92.383,169.951,39.071,157.359
C06150=1040.405,115.886,-92.404,169.953,39.073,157.359
C06151=1040.411,116.135,-92.424,169.955,39.073,157.359
C06152=1040.417,116.384,-92.444,169.957,39.074,157.360
C06153=1040.423,116.633,-92.465,169.959,39.075,157.360
C06154=1040.429,116.882,-92.486,169.962,39.075,157.360
C06155=1040.435,117.131,-92.506,169.964,39.076,157.360
C06156=1040.441,117.380,-92.526,169.965,39.077,157.360
C06157=1040.447,117.629,-92.546,169.967,39.077,157.361
C06158=1040.453,117.879,-92.567,169.969,39.078,157.361
C06159=1040.459,118.128,-92.587,169.971,39.078,157.361
C06160=1040.466,118.377,-92.607,169.974,39.080,157.361
C06161=1040.471,118.626,-92.629,169.976,39.080,157.361
C06162=1040.478,118.875,-92.649,169.978,39.081,157.362
C06163=1040.484,119.124,-92.669,169.980,39.082,157.362
C06164=1040.490,119.373,-92.689,169.982,39.082,157.362
C06165=1040.496,119.623,-92.710,169.984,39.083,157.362
C06166=1040.502,119.871,-92.730,169.987,39.084,157.362
C06167=1040.509,120.120,-92.751,169.989,39.084,157.363
C06168=1040.514,120.369,-92.771,169.990,39.085,157.363
C06169=1040.521,120.619,-92.792,169.992,39.085,157.363
C06170=1040.527,120.867,-92.812,169.994,39.086,157.363
C06171=1040.533,121.117,-92.833,169.996,39.087,157.363
C06172=1040.539,121.366,-92.853,169.999,39.087,157.363
C06173=1040.545,121.615,-92.873,170.001,39.088,157.364
C06174=1040.552,121.864,-92.894,170.003,39.089,157.364
C06175=1040.557,122.113,-92.915,170.005,39.090,157.364
C06176=1040.563,122.362,-92.935,170.007,39.090,157.364
C06177=1040.570,122.612,-92.955,170.010,39.091,157.365
C06178=1040.576,122.860,-92.977,170.012,39.092,157.365
C06179=1040.582,123.110,-92.997,170.014,39.092,157.365
C06180=1040.588,123.359,-93.017,170.016,39.093,157.365
C06181=1040.594,123.608,-93.039,170.018,39.094,157.365
C06182=1040.600,123.857,-93.058,170.020,39.094,157.365
C06183=1040.607,124.106,-93.079,170.022,39.095,157.366
C06184=1040.612,124.355,-93.100,170.025,39.095,157.366
C06185=1040.619,124.604,-93.120,170.027,39.096,157.366
C06186=1040.626,124.889,-93.144,170.029,39.097,157.366
C06187=1040.634,125.176,-93.168,170.031,39.098,157.366
C06188=1040.640,125.462,-93.191,170.033,39.099,157.367
C06189=1040.647,125.747,-93.215,170.037,39.099,157.367
C06190=1040.654,125.996,-93.236,170.039,39.100,157.367
C06191=1040.660,126.246,-93.257,170.041,39.101,157.367
C06192=1040.666,126.495,-93.277,170.043,39.101,157.367
C06193=1040.672,126.744,-93.298,170.045,39.102,157.368
C06194=1040.678,126.993,-93.318,170.048,39.103,157.368
C06195=1040.685,127.241,-93.339,170.049,39.103,157.368
C06196=1040.690,127.491,-93.360,170.051,39.104,157.368
C06197=1040.697,127.739,-93.381,170.053,39.104,157.368
C06198=1040.704,127.989,-93.401,170.055,39.105,157.369
C06199=1040.710,128.237,-93.422,170.057,39.106,157.369
C06200=1040.716,128.487,-93.443,170.059,39.106,157.369
C06201=1040.723,128.736,-93.464,170.062,39.107,157.369
C06202=1040.728,128.985,-93.484,170.064,39.108,157.369
C06203=1040.735,129.234,-93.505,170.066,39.108,157.370
C06204=1040.741,129.483,-93.525,170.068,39.109,157.370
C06205=1040.747,129.732,-93.547,170.070,39.109,157.370
C06206=1040.754,129.981,-93.567,170.073,39.111,157.370
C06207=1040.760,130.230,-93.588,170.075,39.111,157.370
C06208=1040.766,130.479,-93.609,170.077,39.112,157.370
C06209=1040.773,130.728,-93.630,170.079,39.112,157.371
C06210=1040.779,130.977,-93.650,170.081,39.113,157.371
C06211=1040.785,131.226,-93.672,170.083,39.114,157.371
C06212=1040.791,131.476,-93.693,170.085,39.114,157.371
C06213=1040.797,131.724,-93.713,170.088,39.115,157.372
C06214=1040.803,131.974,-93.735,170.090,39.116,157.372
C06215=1040.809,132.223,-93.756,170.092,39.117,157.372
C06216=1040.816,132.472,-93.776,170.094,39.117,157.372
C06217=1040.822,132.721,-93.798,170.096,39.118,157.372
C06218=1040.828,132.970,-93.820,170.099,39.119,157.373
C06219=1040.834,133.219,-93.840,170.101,39.120,157.373
C06220=1040.840,133.468,-93.861,170.103,39.121,157.373
C06221=1040.846,133.717,-93.883,170.105,39.121,157.373
C06222=1040.852,133.966,-93.903,170.107,39.122,157.373
C06223=1040.858,134.215,-93.924,170.110,39.123,157.374
C06224=1040.864,134.464,-93.946,170.112,39.123,157.374
C06225=1040.871,134.713,-93.967,170.114,39.124,157.374
C06226=1040.877,134.962,-93.988,170.116,39.125,157.374
C06227=1040.883,135.212,-94.009,170.118,39.125,157.374
C06228=1040.889,135.460,-94.030,170.121,39.126,157.375
C06229=1040.895,135.709,-94.052,170.123,39.127,157.375
C06230=1040.902,135.958,-94.073,170.125,39.127,157.375
C06231=1040.908,136.207,-94.093,170.127,39.129,157.375
C06232=1040.914,136.456,-94.115,170.129,39.129,157.375
C06233=1040.920,136.706,-94.136,170.132,39.130,157.376
C06234=1040.926,136.954,-94.157,170.134,39.131,157.376
C06235=1040.932,137.203,-94.179,170.136,39.131,157.376
C06236=1040.938,137.452,-94.200,170.138,39.132,157.376
C06237=1040.944,137.702,-94.221,170.140,39.133,157.376
C06238=1040.951,137.950,-94.242,170.142,39.134,157.377
C06239=1040.957,138.199,-94.264,170.145,39.134,157.377
C06240=1040.963,138.449,-94.285,170.147,39.136,157.377
C06241=1040.969,138.698,-94.307,170.149,39.136,157.377
C06242=1040.975,138.946,-94.328,170.151,39.136,157.378
C06243=1040.982,139.195,-94.349,170.154,39.138,157.378
C06244=1040.988,139.444,-94.371,170.157,39.138,157.378
C06245=1040.994,139.694,-94.393,170.159,39.139,157.378
C06246=1040.999,139.942,-94.414,170.161,39.140,157.378
C06247=1041.006,140.191,-94.435,170.163,39.141,157.379
C06248=1041.012,140.440,-94.457,170.165,39.141,157.379
C06249=1041.018,140.690,-94.479,170.168,39.142,157.379
C06250=1041.025,140.975,-94.502,170.170,39.143,157.379
C06251=1041.032,141.261,-94.528,170.172,39.144,157.380
C06252=1041.038,141.547,-94.552,170.175,39.145,157.380
C06253=1041.046,141.832,-94.577,170.178,39.146,157.380
C06254=1041.052,142.081,-94.598,170.180,39.147,157.380
C06255=1041.058,142.330,-94.620,170.182,39.148,157.381
C06256=1041.064,142.579,-94.641,170.184,39.148,157.381
C06257=1041.070,142.828,-94.663,170.186,39.149,157.381
C06258=1041.077,143.077,-94.684,170.189,39.150,157.381
C06259=1041.082,143.326,-94.706,170.191,39.151,157.382
C06260=1041.089,143.574,-94.728,170.193,39.151,157.382
C06261=1041.095,143.824,-94.750,170.195,39.153,157.382
C06262=1041.101,144.073,-94.771,170.197,39.153,157.382
C06263=1041.107,144.322,-94.793,170.200,39.154,157.382
C06264=1041.113,144.571,-94.814,170.202,39.155,157.383
C06265=1041.119,144.820,-94.836,170.204,39.156,157.383
C06266=1041.125,145.069,-94.858,170.206,39.156,157.383
C06267=1041.131,145.318,-94.879,170.209,39.157,157.383
C06268=1041.138,145.567,-94.902,170.212,39.158,157.384
C06269=1041.144,145.816,-94.923,170.214,39.158,157.384
C06270=1041.151,146.065,-94.944,170.216,39.159,157.384
C06271=1041.156,146.313,-94.965,170.218,39.160,157.384
C06272=1041.162,146.563,-94.987,170.220,39.161,157.384
C06273=1041.169,146.811,-95.009,170.223,39.161,157.385
C06274=1041.175,147.060,-95.031,170.225,39.163,157.385
C06275=1041.181,147.310,-95.053,170.227,39.164,157.385
C06276=1041.187,147.559,-95.075,170.229,39.164,157.385
C06277=1041.193,147.808,-95.097,170.231,39.165,157.386
C06278=1041.199,148.057,-95.119,170.234,39.166,157.386
C06279=1041.205,148.305,-95.140,170.236,39.167,157.386
C06280=1041.211,148.555,-95.162,170.238,39.167,157.386
C06281=1041.217,148.803,-95.184,170.240,39.169,157.386
C06282=1041.224,149.052,-95.206,170.244,39.170,157.387
C06283=1041.230,149.302,-95.227,170.246,39.170,157.387
C06284=1041.235,149.551,-95.250,170.248,39.171,157.387
C06285=1041.242,149.800,-95.272,170.250,39.172,157.387
C06286=1041.248,150.049,-95.294,170.252,39.173,157.388
C06287=1041.254,150.298,-95.316,170.255,39.174,157.388
C06288=1041.260,150.546,-95.337,170.257,39.174,157.388
C06289=1041.266,150.795,-95.360,170.259,39.175,157.388
C06290=1041.272,151.044,-95.382,170.261,39.176,157.389
C06291=1041.278,151.293,-95.404,170.263,39.177,157.389
C06292=1041.284,151.542,-95.426,170.266,39.178,157.389
C06293=1041.291,151.791,-95.448,170.268,39.179,157.389
C06294=1041.296,152.040,-95.470,170.271,39.180,157.390
C06295=1041.302,152.289,-95.492,170.273,39.180,157.390
C06296=1041.309,152.538,-95.514,170.276,39.181,157.390
C06297=1041.315,152.787,-95.536,170.278,39.182,157.390
C06298=1041.322,153.036,-95.558,170.280,39.183,157.391
C06299=1041.327,153.285,-95.581,170.282,39.184,157.391
C06300=1041.333,153.534,-95.603,170.284,39.185,157.391
C06301=1041.340,153.783,-95.625,170.287,39.186,157.391
C06302=1041.346,154.031,-95.647,170.289,39.187,157.392
C06303=1041.351,154.281,-95.669,170.291,39.187,157.392
C06304=1041.358,154.530,-95.692,170.294,39.188,157.392
C06305=1041.364,154.779,-95.713,170.297,39.189,157.392
C06306=1041.371,155.027,-95.736,170.299,39.190,157.392
C06307=1041.375,155.276,-95.757,170.301,39.191,157.393
C06308=1041.382,155.525,-95.780,170.303,39.192,157.393
C06309=1041.388,155.774,-95.803,170.305,39.193,157.393
C06310=1041.394,156.023,-95.824,170.308,39.194,157.393
C06311=1041.400,156.271,-95.847,170.310,39.195,157.394
C06312=1041.406,156.520,-95.870,170.312,39.196,157.394
C06313=1041.412,156.770,-95.891,170.315,39.196,157.394
C06314=1041.420,157.055,-95.917,170.318,39.197,157.395
C06315=1041.427,157.341,-95.943,170.320,39.199,157.395
C06316=1041.433,157.626,-95.968,170.323,39.200,157.395
C06317=1041.440,157.911,-95.994,170.325,39.201,157.395
C06318=1041.447,158.160,-96.017,170.329,39.202,157.396
C06319=1041.453,158.409,-96.038,170.331,39.202,157.396
C06320=1041.458,158.658,-96.061,170.333,39.203,157.396
C06321=1041.465,158.906,-96.084,170.335,39.204,157.396
C06322=1041.471,159.156,-96.105,170.337,39.205,157.397
C06323=1041.477,159.404,-96.128,170.340,39.206,157.397
C06324=1041.483,159.653,-96.150,170.342,39.207,157.397
C06325=1041.489,159.902,-96.173,170.345,39.208,157.397
C06326=1041.496,160.152,-96.195,170.347,39.209,157.398
C06327=1041.502,160.401,-96.218,170.350,39.210,157.398
C06328=1041.508,160.649,-96.241,170.352,39.211,157.398
C06329=1041.514,160.898,-96.264,170.354,39.212,157.399
C06330=1041.519,161.147,-96.287,170.356,39.213,157.399
C06331=1041.525,161.396,-96.310,170.359,39.214,157.399
C06332=1041.531,161.645,-96.333,170.361,39.215,157.399
C06333=1041.537,161.893,-96.355,170.364,39.216,157.400
C06334=1041.543,162.142,-96.378,170.366,39.217,157.400
C06335=1041.549,162.392,-96.400,170.369,39.218,157.400
C06336=1041.554,162.641,-96.423,170.371,39.219,157.400
C06337=1041.561,162.889,-96.445,170.373,39.220,157.401
C06338=1041.566,163.138,-96.468,170.376,39.221,157.401
C06339=1041.572,163.387,-96.491,170.378,39.222,157.401
C06340=1041.578,163.636,-96.514,170.380,39.223,157.402
C06341=1041.584,163.885,-96.537,170.383,39.225,157.402
C06342=1041.590,164.134,-96.559,170.386,39.226,157.402
C06343=1041.596,164.382,-96.582,170.388,39.227,157.403
C06344=1041.602,164.631,-96.605,170.390,39.228,157.403
C06345=1041.607,164.880,-96.628,170.392,39.228,157.403
C06346=1041.613,165.129,-96.651,170.395,39.229,157.403
C06347=1041.620,165.378,-96.674,170.398,39.230,157.404
C06348=1041.626,165.627,-96.698,170.400,39.232,157.404
C06349=1041.632,165.876,-96.721,170.402,39.233,157.404
C06350=1041.638,166.125,-96.744,170.405,39.234,157.404
C06351=1041.643,166.373,-96.766,170.407,39.235,157.405
C06352=1041.650,166.622,-96.789,170.409,39.236,157.405
C06353=1041.656,166.871,-96.812,170.412,39.237,157.405
C06354=1041.661,167.120,-96.835,170.415,39.238,157.406
C06355=1041.668,167.369,-96.858,170.417,39.239,157.406
C06356=1041.673,167.618,-96.881,170.419,39.240,157.406
C06357=1041.679,167.867,-96.904,170.422,39.241,157.406
C06358=1041.686,168.115,-96.927,170.424,39.243,157.407
C06359=1041.692,168.364,-96.950,170.427,39.243,157.407
C06360=1041.697,168.613,-96.973,170.429,39.244,157.407
C06361=1041.704,168.863,-96.996,170.431,39.245,157.408
C06362=1041.710,169.104,-97.018,170.434,39.246,157.408
C06363=1041.715,169.347,-97.041,170.436,39.247,157.408
C06364=1041.721,169.590,-97.064,170.438,39.248,157.408
C06365=1041.727,169.832,-97.086,170.442,39.250,157.409
C06366=1041.733,170.074,-97.109,170.444,39.251,157.409
C06367=1041.739,170.317,-97.130,170.446,39.252,157.409
C06368=1041.745,170.560,-97.153,170.448,39.253,157.410
C06369=1041.751,170.803,-97.176,170.451,39.253,157.410
C06370=1041.757,171.051,-97.199,170.453,39.254,157.410
C06371=1041.763,171.299,-97.222,170.456,39.255,157.410
C06372=1041.769,171.548,-97.245,170.458,39.257,157.411
C06373=1041.775,171.798,-97.269,170.461,39.258,157.411
C06374=1041.781,172.047,-97.292,170.463,39.259,157.411
C06375=1041.787,172.295,-97.315,170.466,39.260,157.412
C06376=1041.793,172.544,-97.338,170.468,39.261,157.412
C06377=1041.800,172.793,-97.361,170.471,39.262,157.412
C06378=1041.807,173.090,-97.389,170.474,39.263,157.412
C06379=1041.814,173.388,-97.416,170.477,39.265,157.413
C06380=1041.821,173.686,-97.445,170.480,39.266,157.413
C06381=1041.828,173.983,-97.473,170.483,39.267,157.413
C06382=1041.835,174.232,-97.495,170.485,39.268,157.414
C06383=1041.841,174.481,-97.519,170.487,39.269,157.414
C06384=1041.847,174.730,-97.542,170.491,39.270,157.414
C06385=1041.853,174.978,-97.566,170.493,39.271,157.415
C06386=1041.860,175.228,-97.589,170.495,39.272,157.415
C06387=1041.865,175.476,-97.612,170.499,39.273,157.415
C06388=1041.871,175.725,-97.635,170.501,39.274,157.416
C06389=1041.878,175.974,-97.659,170.503,39.275,157.416
C06390=1041.884,176.222,-97.682,170.505,39.277,157.416
C06391=1041.890,176.471,-97.705,170.509,39.278,157.416
C06392=1041.897,176.720,-97.729,170.511,39.279,157.417
C06393=1041.902,176.969,-97.752,170.513,39.280,157.417
C06394=1041.909,177.218,-97.776,170.517,39.281,157.417
C06395=1041.915,177.467,-97.799,170.519,39.282,157.418
C06396=1041.921,177.715,-97.822,170.521,39.283,157.418
C06397=1041.927,177.965,-97.846,170.523,39.284,157.418
C06398=1041.933,178.213,-97.869,170.527,39.285,157.418
C06399=1041.940,178.462,-97.892,170.529,39.286,157.419
C06400=1041.946,178.711,-97.916,170.531,39.287,157.419
C06401=1041.952,178.960,-97.939,170.534,39.288,157.419
C06402=1041.959,179.209,-97.963,170.537,39.289,157.420
C06403=1041.964,179.457,-97.986,170.539,39.291,157.420
C06404=1041.971,179.706,-98.010,170.542,39.292,157.420
C06405=1041.977,179.955,-98.033,170.545,39.293,157.421
C06406=1041.983,180.204,-98.057,170.547,39.294,157.421
C06407=1041.990,180.453,-98.080,170.550,39.295,157.421
C06408=1041.996,180.702,-98.104,170.552,39.296,157.421
C06409=1042.002,180.950,-98.127,170.555,39.297,157.422
C06410=1042.009,181.199,-98.151,170.558,39.298,157.422
C06411=1042.015,181.448,-98.174,170.560,39.299,157.422
C06412=1042.022,181.697,-98.198,170.562,39.300,157.423
C06413=1042.028,181.945,-98.221,170.566,39.301,157.423
C06414=1042.034,182.195,-98.245,170.568,39.302,157.423
C06415=1042.040,182.443,-98.268,170.570,39.303,157.424
C06416=1042.047,182.692,-98.292,170.574,39.304,157.424
C06417=1042.053,182.940,-98.316,170.576,39.306,157.424
C06418=1042.059,183.190,-98.339,170.579,39.307,157.424
C06419=1042.065,183.438,-98.363,170.581,39.308,157.425
C06420=1042.072,183.687,-98.387,170.584,39.309,157.425
C06421=1042.078,183.935,-98.411,170.587,39.310,157.425
C06422=1042.084,184.185,-98.435,170.589,39.311,157.426
C06423=1042.090,184.433,-98.459,170.592,39.313,157.426
C06424=1042.095,184.682,-98.482,170.595,39.314,157.427
C06425=1042.101,184.931,-98.507,170.597,39.315,157.427
C06426=1042.107,185.180,-98.531,170.600,39.316,157.427
C06427=1042.113,185.429,-98.555,170.603,39.318,157.428
C06428=1042.119,185.677,-98.579,170.605,39.319,157.428
C06429=1042.125,185.926,-98.603,170.608,39.320,157.428
C06430=1042.130,186.175,-98.627,170.611,39.322,157.429
C06431=1042.137,186.424,-98.651,170.613,39.323,157.429
C06432=1042.142,186.673,-98.676,170.615,39.324,157.429
C06433=1042.149,186.922,-98.700,170.619,39.326,157.430
C06434=1042.154,187.170,-98.724,170.621,39.327,157.430
C06435=1042.161,187.419,-98.748,170.624,39.329,157.430
C06436=1042.166,187.668,-98.772,170.627,39.330,157.431
C06437=1042.173,187.917,-98.796,170.629,39.331,157.431
C06438=1042.178,188.165,-98.820,170.632,39.332,157.431
C06439=1042.185,188.414,-98.845,170.635,39.333,157.432
C06440=1042.190,188.662,-98.869,170.637,39.334,157.432
C06441=1042.197,188.911,-98.894,170.639,39.336,157.432
C06442=1042.204,189.195,-98.920,170.643,39.338,157.433
C06443=1042.211,189.480,-98.949,170.646,39.339,157.433
C06444=1042.217,189.765,-98.977,170.650,39.340,157.434
C06445=1042.225,190.049,-99.005,170.652,39.342,157.434
C06446=1042.231,190.297,-99.028,170.655,39.343,157.434
C06447=1042.237,190.546,-99.053,170.658,39.344,157.435
C06448=1042.243,190.795,-99.077,170.660,39.346,157.435
C06449=1042.248,191.044,-99.101,170.663,39.347,157.435
C06450=1042.255,191.292,-99.126,170.666,39.349,157.436
C06451=1042.261,191.541,-99.150,170.669,39.350,157.436
C06452=1042.267,191.790,-99.175,170.671,39.351,157.436
C06453=1042.273,192.039,-99.198,170.674,39.353,157.437
C06454=1042.279,192.288,-99.223,170.677,39.354,157.437
C06455=1042.285,192.536,-99.248,170.679,39.355,157.437
C06456=1042.291,192.785,-99.272,170.683,39.356,157.438
C06457=1042.297,193.034,-99.296,170.685,39.358,157.438
C06458=1042.304,193.282,-99.321,170.687,39.359,157.439
C06459=1042.310,193.531,-99.345,170.691,39.360,157.439
C06460=1042.316,193.780,-99.370,170.693,39.362,157.439
C06461=1042.322,194.029,-99.394,170.696,39.363,157.440
C06462=1042.328,194.277,-99.419,170.699,39.365,157.440
C06463=1042.334,194.526,-99.443,170.702,39.366,157.440
C06464=1042.340,194.775,-99.467,170.704,39.367,157.441
C06465=1042.346,195.023,-99.492,170.708,39.368,157.441
C06466=1042.353,195.272,-99.516,170.710,39.370,157.441
C06467=1042.359,195.521,-99.542,170.712,39.371,157.442
C06468=1042.365,195.770,-99.566,170.716,39.372,157.442
C06469=1042.371,196.018,-99.590,170.718,39.374,157.443
C06470=1042.378,196.267,-99.615,170.721,39.375,157.443
C06471=1042.384,196.516,-99.639,170.724,39.376,157.443
C06472=1042.391,196.764,-99.664,170.727,39.377,157.444
C06473=1042.396,197.013,-99.688,170.729,39.379,157.444
C06474=1042.402,197.262,-99.713,170.733,39.380,157.444
C06475=1042.409,197.511,-99.738,170.735,39.382,157.445
C06476=1042.415,197.760,-99.762,170.738,39.383,157.445
C06477=1042.421,198.008,-99.787,170.741,39.385,157.445
C06478=1042.427,198.257,-99.811,170.744,39.386,157.446
C06479=1042.434,198.505,-99.836,170.746,39.387,157.446
C06480=1042.440,198.755,-99.861,170.750,39.388,157.447
C06481=1042.446,199.003,-99.886,170.752,39.390,157.447
C06482=1042.452,199.251,-99.910,170.755,39.391,157.447
C06483=1042.458,199.500,-99.935,170.758,39.393,157.448
C06484=1042.465,199.748,-99.960,170.761,39.394,157.448
C06485=1042.471,199.998,-99.984,170.764,39.395,157.448
C06486=1042.477,200.246,-100.010,170.767,39.396,157.449
C06487=1042.484,200.495,-100.034,170.769,39.398,157.449
C06488=1042.489,200.743,-100.059,170.773,39.399,157.449
C06489=1042.496,200.992,-100.083,170.775,39.401,157.450
C06490=1042.502,201.241,-100.108,170.778,39.403,157.450
C06491=1042.508,201.490,-100.133,170.781,39.404,157.451
C06492=1042.514,201.739,-100.158,170.784,39.405,157.451
C06493=1042.521,201.988,-100.183,170.786,39.407,157.451
C06494=1042.526,202.236,-100.208,170.790,39.408,157.452
C06495=1042.532,202.484,-100.234,170.792,39.410,157.452
C06496=1042.538,202.734,-100.258,170.796,39.411,157.453
C06497=1042.545,202.982,-100.283,170.798,39.413,157.453
C06498=1042.551,203.231,-100.308,170.801,39.414,157.453
C06499=1042.558,203.479,-100.334,170.804,39.416,157.454
C06500=1042.563,203.727,-100.359,170.807,39.417,157.454
C06501=1042.569,203.977,-100.383,170.810,39.419,157.455
C06502=1042.575,204.225,-100.409,170.813,39.420,157.455
C06503=1042.582,204.474,-100.434,170.815,39.422,157.455
C06504=1042.588,204.723,-100.459,170.819,39.423,157.456
C06505=1042.594,204.971,-100.485,170.822,39.425,157.456
C06506=1042.620,206.023,-100.591,171.095,39.527,157.487
C06507=1042.628,206.315,-100.622,171.097,39.530,157.487
C06508=1042.636,206.607,-100.653,171.100,39.533,157.488
C06509=1042.643,206.899,-100.684,171.102,39.535,157.488
C06510=1042.651,207.192,-100.715,171.105,39.538,157.489
C06511=1042.658,207.440,-100.741,171.107,39.540,157.490
C06512=1042.665,207.688,-100.768,171.109,39.542,157.490
C06513=1042.672,207.937,-100.794,171.111,39.544,157.491
C06514=1042.678,208.186,-100.821,171.114,39.546,157.491
C06515=1042.685,208.434,-100.847,171.115,39.549,157.492
C06516=1042.692,208.683,-100.873,171.118,39.551,157.492
C06517=1042.697,208.931,-100.900,171.120,39.554,157.493
C06518=1042.705,209.180,-100.926,171.122,39.556,157.494
C06519=1042.711,209.428,-100.953,171.125,39.558,157.494
C06520=1042.717,209.677,-100.980,171.126,39.560,157.495
C06521=1042.724,209.925,-101.006,171.129,39.563,157.495
C06522=1042.731,210.174,-101.032,171.131,39.565,157.496
C06523=1042.737,210.423,-101.059,171.133,39.567,157.496
C06524=1042.744,210.671,-101.085,171.135,39.569,157.497
C06525=1042.751,210.920,-101.113,171.138,39.571,157.497
C06526=1042.757,211.168,-101.139,171.139,39.574,157.498
C06527=1042.764,211.416,-101.165,171.142,39.576,157.498
C06528=1042.771,211.666,-101.192,171.144,39.578,157.499
C06529=1042.777,211.914,-101.218,171.146,39.581,157.500
C06530=1042.784,212.163,-101.245,171.149,39.583,157.500
C06531=1042.790,212.410,-101.272,171.150,39.585,157.501
C06532=1042.797,212.659,-101.299,171.153,39.588,157.501
C06533=1042.804,212.908,-101.326,171.155,39.590,157.502
C06534=1042.810,213.156,-101.352,171.157,39.592,157.502
C06535=1042.817,213.404,-101.379,171.159,39.594,157.503
C06536=1042.823,213.653,-101.406,171.162,39.596,157.503
C06537=1042.829,213.902,-101.433,171.163,39.599,157.504
C06538=1042.836,214.151,-101.459,171.166,39.601,157.504
C06539=1042.842,214.398,-101.487,171.169,39.603,157.505
C06540=1042.849,214.647,-101.513,171.170,39.606,157.506
C06541=1042.855,214.895,-101.540,171.173,39.608,157.506
C06542=1042.863,215.144,-101.567,171.175,39.610,157.507
C06543=1042.869,215.393,-101.594,171.177,39.613,157.507
C06544=1042.875,215.641,-101.621,171.179,39.615,157.508
C06545=1042.882,215.889,-101.648,171.182,39.617,157.508
C06546=1042.889,216.138,-101.675,171.184,39.619,157.509
C06547=1042.895,216.386,-101.701,171.186,39.621,157.509
C06548=1042.902,216.635,-101.729,171.188,39.624,157.510
C06549=1042.909,216.883,-101.755,171.191,39.626,157.511
C06550=1042.915,217.131,-101.782,171.193,39.628,157.511
C06551=1042.921,217.380,-101.809,171.195,39.630,157.512
C06552=1042.928,217.629,-101.836,171.198,39.633,157.512
C06553=1042.935,217.877,-101.864,171.200,39.635,157.513
C06554=1042.942,218.125,-101.890,171.202,39.637,157.513
C06555=1042.948,218.374,-101.917,171.204,39.639,157.514
C06556=1042.955,218.623,-101.944,171.207,39.641,157.514
C06557=1042.962,218.871,-101.971,171.209,39.644,157.515
C06558=1042.968,219.119,-101.998,171.211,39.646,157.515
C06559=1042.975,219.368,-102.025,171.214,39.648,157.516
C06560=1042.982,219.617,-102.052,171.216,39.651,157.517
C06561=1042.989,219.865,-102.079,171.219,39.652,157.517
C06562=1042.995,220.113,-102.106,171.220,39.655,157.518
C06563=1043.003,220.411,-102.139,171.223,39.658,157.518
C06564=1043.011,220.709,-102.172,171.226,39.660,157.519
C06565=1043.019,221.006,-102.204,171.229,39.663,157.520
C06566=1043.026,221.305,-102.237,171.232,39.666,157.520
C06567=1043.033,221.554,-102.264,171.233,39.668,157.521
C06568=1043.039,221.801,-102.292,171.236,39.670,157.521
C06569=1043.046,222.050,-102.318,171.239,39.672,157.522
C06570=1043.053,222.298,-102.346,171.241,39.675,157.523
C06571=1043.059,222.547,-102.374,171.243,39.677,157.523
C06572=1043.065,222.795,-102.400,171.245,39.679,157.524
C06573=1043.072,223.044,-102.428,171.248,39.682,157.524
C06574=1043.078,223.292,-102.456,171.250,39.684,157.525
C06575=1043.085,223.541,-102.483,171.253,39.686,157.525
C06576=1043.092,223.789,-102.510,171.254,39.688,157.526
C06577=1043.098,224.037,-102.537,171.257,39.690,157.526
C06578=1043.105,224.286,-102.565,171.259,39.693,157.527
C06579=1043.112,224.534,-102.593,171.262,39.695,157.528
C06580=1043.118,224.783,-102.620,171.265,39.697,157.528
C06581=1043.125,225.032,-102.647,171.266,39.699,157.529
C06582=1043.131,225.279,-102.675,171.269,39.702,157.529
C06583=1043.138,225.527,-102.702,171.271,39.704,157.530
C06584=1043.145,225.776,-102.729,171.274,39.706,157.530
C06585=1043.151,226.025,-102.757,171.276,39.708,157.531
C06586=1043.158,226.273,-102.784,171.278,39.710,157.531
C06587=1043.165,226.522,-102.812,171.280,39.713,157.532
C06588=1043.171,226.770,-102.840,171.283,39.715,157.533
C06589=1043.177,227.018,-102.867,171.286,39.717,157.533
C06590=1043.184,227.267,-102.894,171.288,39.719,157.534
C06591=1043.190,227.515,-102.922,171.291,39.722,157.534
C06592=1043.198,227.764,-102.949,171.292,39.724,157.535
C06593=1043.205,228.012,-102.977,171.295,39.726,157.535
C06594=1043.211,228.260,-103.005,171.297,39.728,157.536
C06595=1043.218,228.509,-103.032,171.300,39.730,157.536
C06596=1043.225,228.757,-103.060,171.303,39.733,157.537
C06597=1043.231,229.006,-103.088,171.305,39.735,157.538
C06598=1043.237,229.254,-103.115,171.308,39.737,157.538
C06599=1043.244,229.502,-103.143,171.309,39.739,157.539
C06600=1043.250,229.751,-103.171,171.312,39.742,157.539
C06601=1043.257,229.999,-103.199,171.314,39.744,157.540
C06602=1043.263,230.248,-103.227,171.317,39.746,157.540
C06603=1043.270,230.496,-103.254,171.320,39.749,157.541
C06604=1043.277,230.744,-103.282,171.322,39.751,157.542
C06605=1043.283,230.993,-103.310,171.325,39.753,157.542
C06606=1043.290,231.241,-103.338,171.326,39.755,157.543
C06607=1043.297,231.490,-103.365,171.329,39.757,157.543
C06608=1043.303,231.738,-103.393,171.331,39.759,157.544
C06609=1043.309,231.986,-103.421,171.334,39.762,157.544
C06610=1043.315,232.235,-103.449,171.336,39.764,157.545
C06611=1043.322,232.483,-103.477,171.339,39.766,157.545
C06612=1043.329,232.731,-103.505,171.342,39.768,157.546
C06613=1043.335,232.980,-103.533,171.344,39.771,157.547
C06614=1043.342,233.228,-103.561,171.347,39.773,157.547
C06615=1043.348,233.477,-103.589,171.348,39.775,157.548
C06616=1043.355,233.725,-103.616,171.351,39.778,157.548
C06617=1043.361,233.973,-103.645,171.353,39.780,157.549
C06618=1043.368,234.222,-103.673,171.356,39.782,157.549
C06619=1043.376,234.511,-103.706,171.359,39.785,157.550
C06620=1043.384,234.803,-103.739,171.362,39.787,157.551
C06621=1043.392,235.093,-103.771,171.365,39.790,157.551
C06622=1043.399,235.383,-103.804,171.368,39.793,157.552
C06623=1043.406,235.631,-103.832,171.370,39.795,157.553
C06624=1043.412,235.880,-103.861,171.373,39.797,157.553
C06625=1043.418,236.128,-103.888,171.375,39.799,157.554
C06626=1043.425,236.376,-103.917,171.378,39.801,157.554
C06627=1043.432,236.625,-103.945,171.381,39.804,157.555
C06628=1043.438,236.873,-103.973,171.383,39.806,157.556
C06629=1043.445,237.121,-104.001,171.386,39.808,157.556
C06630=1043.451,237.370,-104.029,171.388,39.810,157.557
C06631=1043.458,237.618,-104.057,171.391,39.813,157.557
C06632=1043.464,237.866,-104.086,171.394,39.815,157.558
C06633=1043.472,238.115,-104.114,171.396,39.817,157.558
C06634=1043.479,238.363,-104.142,171.399,39.820,157.559
C06635=1043.485,238.612,-104.171,171.401,39.822,157.560
C06636=1043.491,238.860,-104.198,171.403,39.824,157.560
C06637=1043.498,239.108,-104.227,171.405,39.826,157.561
C06638=1043.504,239.357,-104.255,171.408,39.829,157.561
C06639=1043.511,239.605,-104.284,171.411,39.831,157.562
C06640=1043.517,239.853,-104.312,171.413,39.833,157.562
C06641=1043.524,240.101,-104.340,171.416,39.835,157.563
C06642=1043.531,240.350,-104.368,171.418,39.837,157.563
C06643=1043.537,240.598,-104.397,171.421,39.839,157.564
C06644=1043.544,240.847,-104.425,171.423,39.842,157.565
C06645=1043.551,241.095,-104.454,171.426,39.844,157.565
C06646=1043.557,241.344,-104.482,171.429,39.846,157.566
C06647=1043.564,241.591,-104.511,171.431,39.848,157.566
C06648=1043.571,241.839,-104.540,171.434,39.851,157.567
C06649=1043.576,242.088,-104.568,171.436,39.853,157.568
C06650=1043.583,242.336,-104.596,171.439,39.855,157.568
C06651=1043.589,242.585,-104.625,171.441,39.857,157.569
C06652=1043.596,242.833,-104.653,171.444,39.860,157.569
C06653=1043.603,243.081,-104.682,171.447,39.862,157.570
C06654=1043.609,243.330,-104.712,171.449,39.864,157.570
C06655=1043.616,243.578,-104.739,171.452,39.866,157.571
C06656=1043.622,243.826,-104.768,171.454,39.869,157.572
C06657=1043.629,244.074,-104.797,171.457,39.872,157.572
C06658=1043.635,244.323,-104.825,171.461,39.874,157.573
C06659=1043.642,244.571,-104.854,171.463,39.876,157.573
C06660=1043.649,244.819,-104.883,171.466,39.878,157.574
C06661=1043.655,245.068,-104.912,171.469,39.881,157.575
C06662=1043.662,245.316,-104.940,171.471,39.883,157.575
C06663=1043.668,245.564,-104.969,171.474,39.885,157.576
C06664=1043.675,245.812,-104.998,171.476,39.887,157.576
C06665=1043.681,246.060,-105.027,171.479,39.890,157.577
C06666=1043.687,246.309,-105.056,171.481,39.892,157.578
C06667=1043.693,246.557,-105.085,171.484,39.894,157.578
C06668=1043.701,246.805,-105.114,171.487,39.896,157.579
C06669=1043.707,247.053,-105.143,171.489,39.899,157.579
C06670=1043.713,247.302,-105.171,171.492,39.901,157.580
C06671=1043.719,247.550,-105.200,171.495,39.904,157.581
C06672=1043.726,247.798,-105.229,171.497,39.906,157.581
C06673=1043.732,248.046,-105.258,171.500,39.908,157.582
C06674=1043.739,248.295,-105.288,171.502,39.910,157.582
C06675=1043.746,248.579,-105.321,171.506,39.913,157.583
C06676=1043.754,248.864,-105.354,171.509,39.915,157.584
C06677=1043.761,249.148,-105.387,171.511,39.918,157.584
C06678=1043.768,249.433,-105.420,171.515,39.921,157.585
C06679=1043.775,249.682,-105.449,171.518,39.923,157.586
C06680=1043.782,249.930,-105.478,171.520,39.926,157.586
C06681=1043.788,250.177,-105.508,171.523,39.928,157.587
C06682=1043.794,250.425,-105.537,171.526,39.930,157.587
C06683=1043.801,250.674,-105.567,171.528,39.932,157.588
C06684=1043.807,250.922,-105.596,171.531,39.935,157.589
C06685=1043.814,251.170,-105.624,171.533,39.937,157.589
C06686=1043.821,251.418,-105.653,171.536,39.940,157.590
C06687=1043.827,251.667,-105.683,171.540,39.942,157.590
C06688=1043.834,251.915,-105.712,171.542,39.944,157.591
C06689=1043.840,252.164,-105.741,171.545,39.946,157.592
C06690=1043.847,252.412,-105.771,171.547,39.949,157.592
C06691=1043.853,252.660,-105.800,171.550,39.951,157.593
C06692=1043.860,252.908,-105.829,171.553,39.953,157.593
C06693=1043.867,253.157,-105.858,171.555,39.955,157.594
C06694=1043.873,253.405,-105.887,171.559,39.958,157.595
C06695=1043.880,253.653,-105.916,171.562,39.960,157.595
C06696=1043.887,253.901,-105.946,171.564,39.963,157.596
C06697=1043.893,254.149,-105.975,171.567,39.965,157.596
C06698=1043.899,254.397,-106.004,171.569,39.967,157.597
C06699=1043.906,254.646,-106.033,171.572,39.969,157.598
C06700=1043.913,254.894,-106.063,171.575,39.971,157.598
C06701=1043.919,255.142,-106.092,171.578,39.974,157.599
C06702=1043.926,255.391,-106.122,171.581,39.976,157.599
C06703=1043.932,255.638,-106.151,171.583,39.978,157.600
C06704=1043.939,255.887,-106.181,171.586,39.980,157.601
C06705=1043.946,256.135,-106.210,171.589,39.983,157.601
C06706=1043.952,256.383,-106.240,171.592,39.985,157.602
C06707=1043.960,256.631,-106.268,171.595,39.988,157.602
C06708=1043.966,256.879,-106.297,171.598,39.990,157.603
C06709=1043.973,257.127,-106.328,171.600,39.992,157.604
C06710=1043.979,257.376,-106.357,171.603,39.994,157.604
C06711=1043.986,257.624,-106.386,171.606,39.996,157.605
C06712=1043.993,257.872,-106.416,171.609,39.999,157.605
C06713=1043.999,258.120,-106.445,171.612,40.001,157.606
C06714=1044.006,258.368,-106.475,171.614,40.003,157.607
C06715=1044.012,258.616,-106.504,171.618,40.005,157.607
C06716=1044.020,258.865,-106.534,171.620,40.008,157.608
C06717=1044.026,259.113,-106.563,171.623,40.010,157.608
C06718=1044.033,259.362,-106.592,171.626,40.013,157.609
C06719=1044.039,259.609,-106.622,171.629,40.015,157.610
C06720=1044.046,259.858,-106.652,171.632,40.017,157.610
C06721=1044.053,260.105,-106.681,171.635,40.019,157.611
C06722=1044.060,260.354,-106.712,171.637,40.021,157.611
C06723=1044.066,260.602,-106.741,171.641,40.024,157.612
C06724=1044.073,260.850,-106.771,171.643,40.026,157.613
C06725=1044.079,261.098,-106.800,171.646,40.028,157.613
C06726=1044.087,261.346,-106.829,171.649,40.030,157.614
C06727=1044.094,261.595,-106.859,171.652,40.032,157.614
C06728=1044.101,261.842,-106.888,171.655,40.035,157.615
C06729=1044.108,262.091,-106.918,171.657,40.037,157.616
C06730=1044.114,262.339,-106.948,171.661,40.040,157.616
C06731=1044.121,262.622,-106.982,171.664,40.042,157.617
C06732=1044.129,262.905,-107.016,171.668,40.045,157.618
C06733=1044.136,263.189,-107.050,171.670,40.047,157.618
C06734=1044.144,263.471,-107.084,171.674,40.050,157.619
C06735=1044.150,263.720,-107.115,171.677,40.052,157.620
C06736=1044.157,263.967,-107.145,171.679,40.055,157.620
C06737=1044.164,264.216,-107.175,171.683,40.057,157.621
C06738=1044.170,264.463,-107.205,171.686,40.060,157.622
C06739=1044.177,264.712,-107.235,171.688,40.062,157.622
C06740=1044.184,264.961,-107.265,171.692,40.065,157.623
C06741=1044.190,265.208,-107.295,171.695,40.067,157.624
C06742=1044.197,265.457,-107.325,171.697,40.069,157.624
C06743=1044.203,265.704,-107.355,171.700,40.071,157.625
C06744=1044.210,265.953,-107.386,171.704,40.074,157.626
C06745=1044.216,266.200,-107.415,171.706,40.076,157.626
C06746=1044.223,266.448,-107.445,171.709,40.078,157.627
C06747=1044.230,266.697,-107.476,171.712,40.081,157.627
C06748=1044.236,266.944,-107.506,171.715,40.083,157.628
C06749=1044.243,267.193,-107.535,171.718,40.086,157.629
C06750=1044.250,267.442,-107.566,171.721,40.088,157.629
C06751=1044.256,267.689,-107.596,171.724,40.090,157.630
C06752=1044.263,267.938,-107.626,171.727,40.093,157.631
C06753=1044.269,268.185,-107.656,171.730,40.095,157.631
C06754=1044.276,268.434,-107.687,171.733,40.097,157.632
C06755=1044.283,268.681,-107.718,171.736,40.100,157.632
C06756=1044.290,268.929,-107.748,171.739,40.102,157.633
C06757=1044.296,269.177,-107.778,171.742,40.104,157.634
C06758=1044.303,269.426,-107.808,171.745,40.107,157.634
C06759=1044.309,269.673,-107.839,171.748,40.109,157.635
C06760=1044.316,269.922,-107.869,171.751,40.112,157.636
C06761=1044.323,270.170,-107.900,171.754,40.114,157.636
C06762=1044.328,270.418,-107.930,171.757,40.116,157.637
C06763=1044.335,270.666,-107.960,171.760,40.119,157.638
C06764=1044.342,270.914,-107.991,171.764,40.121,157.638
C06765=1044.349,271.162,-108.021,171.766,40.124,157.639
C06766=1044.355,271.410,-108.052,171.769,40.126,157.639
C06767=1044.362,271.658,-108.082,171.773,40.129,157.640
C06768=1044.368,271.906,-108.112,171.775,40.131,157.641
C06769=1044.376,272.154,-108.143,171.778,40.133,157.641
C06770=1044.382,272.402,-108.174,171.782,40.136,157.642
C06771=1044.388,272.650,-108.204,171.784,40.138,157.643
C06772=1044.395,272.898,-108.235,171.788,40.141,157.643
C06773=1044.402,273.146,-108.266,171.791,40.143,157.644
C06774=1044.408,273.395,-108.297,171.793,40.145,157.645
C06775=1044.415,273.642,-108.327,171.797,40.148,157.645
C06776=1044.421,273.890,-108.358,171.800,40.150,157.646
C06777=1044.428,274.139,-108.389,171.804,40.153,157.647
C06778=1044.435,274.386,-108.419,171.806,40.155,157.647
C06779=1044.441,274.634,-108.450,171.810,40.158,157.648
C06780=1044.448,274.882,-108.481,171.813,40.160,157.649
C06781=1044.455,275.130,-108.511,171.815,40.162,157.649
C06782=1044.461,275.379,-108.542,171.819,40.165,157.650
C06783=1044.468,275.626,-108.573,171.822,40.167,157.651
C06784=1044.474,275.874,-108.604,171.825,40.170,157.651
C06785=1044.481,276.122,-108.635,171.828,40.172,157.652
C06786=1044.488,276.371,-108.665,171.832,40.175,157.653
C06787=1044.495,276.658,-108.702,171.834,40.178,157.653
C06788=1044.504,276.945,-108.738,171.838,40.180,157.654
C06789=1044.510,277.233,-108.773,171.842,40.183,157.655
C06790=1044.519,277.521,-108.809,171.846,40.186,157.656
C06791=1044.525,277.768,-108.840,171.849,40.189,157.656
C06792=1044.532,278.016,-108.871,171.852,40.191,157.657
C06793=1044.539,278.265,-108.901,171.855,40.193,157.658
C06794=1044.545,278.513,-108.933,171.859,40.196,157.658
C06795=1044.552,278.760,-108.964,171.861,40.198,157.659
C06796=1044.558,279.009,-108.995,171.865,40.200,157.660
C06797=1044.565,279.256,-109.026,171.868,40.203,157.660
C06798=1044.571,279.504,-109.057,171.871,40.205,157.661
C06799=1044.578,279.753,-109.088,171.874,40.208,157.662
C06800=1044.584,280.000,-109.120,171.878,40.211,157.663
C06801=1044.591,280.248,-109.151,171.881,40.213,157.663
C06802=1044.598,280.496,-109.182,171.884,40.216,157.664
C06803=1044.605,280.744,-109.214,171.887,40.218,157.665
C06804=1044.610,280.992,-109.244,171.891,40.221,157.665
C06805=1044.617,281.240,-109.276,171.894,40.224,157.666
C06806=1044.624,281.488,-109.307,171.897,40.226,157.667
C06807=1044.631,281.736,-109.339,171.900,40.228,157.667
C06808=1044.637,281.984,-109.370,171.904,40.231,157.668
C06809=1044.644,282.232,-109.401,171.906,40.233,157.669
C06810=1044.651,282.479,-109.433,171.910,40.236,157.669
C06811=1044.657,282.728,-109.464,171.913,40.238,157.670
C06812=1044.664,282.976,-109.495,171.917,40.241,157.671
C06813=1044.671,283.224,-109.526,171.919,40.243,157.671
C06814=1044.677,283.472,-109.558,171.923,40.246,157.672
C06815=1044.684,283.720,-109.589,171.926,40.249,157.673
C06816=1044.691,283.967,-109.621,171.929,40.251,157.674
C06817=1044.698,284.215,-109.652,171.933,40.254,157.674
C06818=1044.704,284.463,-109.684,171.936,40.256,157.675
C06819=1044.711,284.711,-109.715,171.940,40.258,157.676
C06820=1044.718,284.959,-109.746,171.942,40.261,157.676
C06821=1044.724,285.207,-109.778,171.946,40.263,157.677
C06822=1044.731,285.455,-109.809,171.949,40.266,157.678
C06823=1044.738,285.703,-109.841,171.953,40.269,157.678
C06824=1044.745,285.951,-109.872,171.956,40.271,157.679
C06825=1044.751,286.199,-109.904,171.959,40.274,157.680
C06826=1044.758,286.446,-109.936,171.963,40.276,157.681
C06827=1044.765,286.694,-109.967,171.965,40.279,157.681
C06828=1044.772,286.942,-109.999,171.969,40.281,157.682
C06829=1044.779,287.190,-110.030,171.973,40.284,157.683
C06830=1044.785,287.437,-110.062,171.976,40.286,157.683
C06831=1044.791,287.686,-110.094,171.979,40.289,157.684
C06832=1044.798,287.933,-110.126,171.982,40.292,157.685
C06833=1044.805,288.181,-110.157,171.986,40.294,157.686
C06834=1044.812,288.429,-110.189,171.990,40.296,157.686
C06835=1044.818,288.677,-110.221,171.992,40.299,157.687
C06836=1044.825,288.924,-110.253,171.996,40.302,157.688
C06837=1044.831,289.172,-110.284,171.999,40.305,157.688
C06838=1044.838,289.420,-110.316,172.003,40.307,157.689
C06839=1044.845,289.668,-110.349,172.006,40.310,157.690
C06840=1044.852,289.916,-110.380,172.009,40.312,157.691
C06841=1044.859,290.164,-110.412,172.013,40.315,157.691
C06842=1044.865,290.412,-110.444,172.017,40.318,157.692
C06843=1044.873,290.711,-110.482,172.021,40.320,157.693
C06844=1044.881,291.011,-110.521,172.025,40.324,157.694
C06845=1044.889,291.309,-110.560,172.028,40.327,157.695
C06846=1044.897,291.609,-110.599,172.032,40.330,157.695
C06847=1044.904,291.856,-110.631,172.036,40.333,157.696
C06848=1044.911,292.104,-110.662,172.040,40.336,157.697
C06849=1044.917,292.352,-110.695,172.043,40.338,157.698
C06850=1044.924,292.600,-110.726,172.046,40.340,157.698
C06851=1044.931,292.848,-110.759,172.050,40.343,157.699
C06852=1044.937,293.096,-110.791,172.053,40.346,157.700
C06853=1044.944,293.343,-110.823,172.057,40.349,157.701
C06854=1044.951,293.591,-110.854,172.061,40.351,157.701
C06855=1044.957,293.839,-110.887,172.063,40.354,157.702
C06856=1044.965,294.087,-110.919,172.067,40.356,157.703
C06857=1044.971,294.335,-110.952,172.071,40.359,157.704
C06858=1044.978,294.582,-110.984,172.074,40.362,157.704
C06859=1044.984,294.830,-111.016,172.077,40.364,157.705
C06860=1044.991,295.078,-111.048,172.081,40.367,157.706
C06861=1044.998,295.326,-111.081,172.085,40.370,157.707
C06862=1045.005,295.573,-111.113,172.088,40.372,157.707
C06863=1045.011,295.821,-111.145,172.092,40.375,157.708
C06864=1045.018,296.069,-111.177,172.095,40.378,157.709
C06865=1045.025,296.317,-111.211,172.098,40.381,157.710
C06866=1045.031,296.565,-111.243,172.102,40.383,157.710
C06867=1045.038,296.812,-111.276,172.106,40.386,157.711
C06868=1045.045,297.059,-111.308,172.110,40.389,157.712
C06869=1045.051,297.308,-111.340,172.113,40.392,157.713
C06870=1045.057,297.556,-111.373,172.116,40.395,157.713
C06871=1045.064,297.804,-111.406,172.120,40.397,157.714
C06872=1045.070,298.051,-111.439,172.123,40.400,157.715
C06873=1045.077,298.298,-111.471,172.127,40.403,157.716
C06874=1045.084,298.547,-111.504,172.131,40.406,157.717
C06875=1045.090,298.794,-111.537,172.134,40.408,157.717
C06876=1045.097,299.042,-111.570,172.137,40.412,157.718
C06877=1045.104,299.289,-111.602,172.141,40.414,157.719
C06878=1045.110,299.538,-111.635,172.145,40.417,157.720
C06879=1045.117,299.785,-111.668,172.149,40.420,157.720
C06880=1045.123,300.033,-111.700,172.152,40.422,157.721
C06881=1045.130,300.281,-111.733,172.155,40.425,157.722
C06882=1045.136,300.529,-111.766,172.159,40.428,157.723
C06883=1045.144,300.775,-111.799,172.163,40.431,157.724
C06884=1045.150,301.024,-111.832,172.166,40.434,157.724
C06885=1045.157,301.271,-111.865,172.170,40.436,157.725
C06886=1045.163,301.519,-111.898,172.174,40.439,157.726
C06887=1045.170,301.767,-111.931,172.177,40.442,157.727
C06888=1045.177,302.014,-111.963,172.181,40.445,157.728
C06889=1045.184,302.262,-111.997,172.184,40.448,157.728
C06890=1045.190,302.510,-112.029,172.188,40.450,157.729
C06891=1045.197,302.757,-112.062,172.192,40.453,157.730
C06892=1045.204,303.005,-112.095,172.196,40.456,157.731
C06893=1045.210,303.253,-112.128,172.200,40.459,157.732
C06894=1045.218,303.500,-112.161,172.203,40.462,157.732
C06895=1045.224,303.748,-112.194,172.206,40.464,157.733
C06896=1045.230,303.996,-112.227,172.210,40.467,157.734
C06897=1045.238,304.243,-112.261,172.214,40.470,157.735
C06898=1045.244,304.491,-112.293,172.218,40.473,157.736
C06899=1045.253,304.807,-112.336,172.223,40.477,157.737
C06900=1045.262,305.122,-112.378,172.227,40.480,157.737
C06901=1045.270,305.438,-112.420,172.232,40.484,157.739
C06902=1045.279,305.754,-112.462,172.237,40.487,157.740
C06903=1045.286,306.001,-112.495,172.240,40.490,157.740
C06904=1045.293,306.249,-112.529,172.244,40.493,157.741
C06905=1045.299,306.496,-112.562,172.248,40.496,157.742
C06906=1045.307,306.744,-112.595,172.252,40.499,157.743
C06907=1045.314,306.991,-112.628,172.255,40.501,157.744
C06908=1045.321,307.239,-112.661,172.259,40.504,157.744
C06909=1045.327,307.486,-112.695,172.263,40.507,157.745
C06910=1045.334,307.735,-112.728,172.267,40.510,157.746
C06911=1045.341,307.982,-112.761,172.271,40.513,157.747
C06912=1045.348,308.230,-112.794,172.275,40.516,157.748
C06913=1045.355,308.478,-112.828,172.278,40.519,157.748
C06914=1045.362,308.725,-112.860,172.281,40.521,157.749
C06915=1045.369,308.973,-112.894,172.285,40.525,157.750
C06916=1045.376,309.220,-112.928,172.289,40.527,157.751
C06917=1045.382,309.468,-112.961,172.293,40.530,157.752
C06918=1045.390,309.715,-112.994,172.297,40.533,157.753
C06919=1045.397,309.963,-113.028,172.301,40.536,157.753
C06920=1045.403,310.211,-113.061,172.305,40.539,157.754
C06921=1045.410,310.458,-113.095,172.309,40.542,157.755
C06922=1045.418,310.706,-113.129,172.312,40.544,157.756
C06923=1045.424,310.954,-113.161,172.316,40.548,157.757
C06924=1045.432,311.201,-113.195,172.320,40.550,157.758
C06925=1045.439,311.449,-113.228,172.324,40.553,157.758
C06926=1045.446,311.696,-113.262,172.328,40.556,157.759
C06927=1045.452,311.944,-113.295,172.332,40.559,157.760
C06928=1045.460,312.192,-113.329,172.336,40.562,157.761
C06929=1045.467,312.439,-113.363,172.340,40.565,157.762
C06930=1045.474,312.687,-113.397,172.344,40.568,157.763
C06931=1045.480,312.934,-113.431,172.348,40.571,157.764
C06932=1045.487,313.182,-113.464,172.352,40.574,157.764
C06933=1045.494,313.430,-113.499,172.356,40.577,157.765
C06934=1045.500,313.677,-113.532,172.360,40.580,157.766
C06935=1045.507,313.925,-113.567,172.363,40.583,157.767
C06936=1045.514,314.173,-113.601,172.367,40.586,157.768
C06937=1045.520,314.420,-113.634,172.371,40.589,157.769
C06938=1045.527,314.668,-113.668,172.375,40.592,157.770
C06939=1045.534,314.915,-113.702,172.379,40.595,157.770
C06940=1045.540,315.163,-113.736,172.383,40.598,157.771
C06941=1045.547,315.410,-113.771,172.387,40.602,157.772
C06942=1045.554,315.658,-113.805,172.391,40.605,157.773
C06943=1045.561,315.905,-113.839,172.395,40.608,157.774
C06944=1045.568,316.153,-113.873,172.399,40.611,157.775
C06945=1045.574,316.400,-113.907,172.403,40.614,157.776
C06946=1045.581,316.648,-113.942,172.407,40.617,157.777
C06947=1045.588,316.895,-113.976,172.411,40.620,157.778
C06948=1045.595,317.143,-114.010,172.415,40.624,157.779
C06949=1045.602,317.391,-114.044,172.419,40.626,157.779
C06950=1045.608,317.638,-114.079,172.423,40.629,157.780
C06951=1045.615,317.885,-114.113,172.427,40.633,157.781
C06952=1045.622,318.133,-114.147,172.431,40.636,157.782
C06953=1045.629,318.380,-114.182,172.435,40.639,157.783
C06954=1045.636,318.628,-114.216,172.439,40.642,157.784
C06955=1045.644,318.948,-114.261,172.444,40.646,157.785
C06956=1045.653,319.269,-114.305,172.449,40.650,157.786
C06957=1045.662,319.588,-114.349,172.454,40.654,157.787
C06958=1045.671,319.909,-114.394,172.460,40.658,157.789
C06959=1045.678,320.156,-114.428,172.464,40.661,157.789
C06960=1045.685,320.404,-114.463,172.468,40.665,157.790
C06961=1045.692,320.651,-114.497,172.472,40.668,157.791
C06962=1045.699,320.899,-114.532,172.476,40.671,157.792
C06963=1045.706,321.147,-114.567,172.481,40.674,157.793
C06964=1045.713,321.394,-114.601,172.485,40.677,157.794
C06965=1045.720,321.642,-114.636,172.489,40.681,157.795
C06966=1045.727,321.889,-114.670,172.493,40.684,157.796
C06967=1045.734,322.137,-114.705,172.497,40.687,157.797
C06968=1045.741,322.384,-114.739,172.501,40.690,157.798
C06969=1045.748,322.632,-114.774,172.505,40.693,157.799
C06970=1045.755,322.879,-114.808,172.509,40.696,157.800
C06971=1045.762,323.126,-114.843,172.514,40.699,157.800
C06972=1045.768,323.374,-114.878,172.518,40.703,157.802
C06973=1045.776,323.621,-114.912,172.522,40.706,157.802
C06974=1045.783,323.869,-114.947,172.526,40.709,157.803
C06975=1045.790,324.116,-114.981,172.530,40.713,157.804
C06976=1045.796,324.364,-115.016,172.534,40.716,157.805
C06977=1045.803,324.611,-115.051,172.539,40.719,157.806
C06978=1045.811,324.859,-115.086,172.543,40.722,157.807
C06979=1045.818,325.106,-115.121,172.547,40.725,157.808
C06980=1045.825,325.354,-115.155,172.551,40.728,157.809
C06981=1045.832,325.601,-115.190,172.555,40.732,157.810
C06982=1045.839,325.849,-115.226,172.560,40.735,157.811
C06983=1045.846,326.096,-115.260,172.564,40.738,157.812
C06984=1045.854,326.344,-115.296,172.568,40.741,157.813
C06985=1045.861,326.591,-115.330,172.572,40.745,157.814
C06986=1045.868,326.839,-115.365,172.577,40.748,157.815
C06987=1045.874,327.086,-115.400,172.581,40.751,157.816
C06988=1045.883,327.334,-115.435,172.585,40.754,157.817
C06989=1045.889,327.581,-115.470,172.589,40.758,157.817
C06990=1045.897,327.828,-115.504,172.594,40.761,157.818
C06991=1045.904,328.076,-115.539,172.598,40.764,157.820
C06992=1045.911,328.324,-115.575,172.602,40.768,157.820
C06993=1045.919,328.571,-115.609,172.606,40.771,157.821
C06994=1045.925,328.818,-115.645,172.611,40.774,157.822
C06995=1045.933,329.066,-115.680,172.615,40.777,157.823
C06996=1045.940,329.313,-115.715,172.620,40.781,157.824
C06997=1045.947,329.560,-115.750,172.625,40.784,157.825
C06998=1045.954,329.807,-115.786,172.629,40.787,157.826
C06999=1045.961,330.055,-115.821,172.633,40.791,157.827
C07000=1045.968,330.303,-115.856,172.637,40.794,157.828
C07001=1045.975,330.550,-115.892,172.642,40.798,157.829
C07002=1045.982,330.797,-115.927,172.646,40.801,157.830
C07003=1045.989,331.045,-115.963,172.650,40.805,157.831
C07004=1045.996,331.292,-115.998,172.654,40.808,157.832
C07005=1046.003,331.539,-116.034,172.659,40.812,157.833
C07006=1046.011,331.787,-116.069,172.663,40.815,157.834
C07007=1046.018,332.034,-116.105,172.668,40.819,157.835
C07008=1046.024,332.281,-116.140,172.673,40.822,157.836
C07009=1046.032,332.529,-116.176,172.677,40.825,157.837
C07010=1046.039,332.776,-116.212,172.681,40.829,157.838
C07011=1046.047,333.091,-116.257,172.687,40.833,157.840
C07012=1046.057,333.407,-116.303,172.693,40.837,157.841
C07013=1046.065,333.722,-116.348,172.698,40.842,157.842
C07014=1046.075,334.037,-116.394,172.704,40.847,157.844
C07015=1046.082,334.285,-116.429,172.709,40.850,157.845
C07016=1046.089,334.532,-116.465,172.713,40.853,157.846
C07017=1046.096,334.779,-116.500,172.717,40.857,157.847
C07018=1046.104,335.027,-116.536,172.722,40.860,157.848
C07019=1046.111,335.274,-116.572,172.726,40.864,157.849
C07020=1046.118,335.522,-116.608,172.731,40.868,157.850
C07021=1046.125,335.768,-116.644,172.736,40.871,157.851
C07022=1046.132,336.016,-116.680,172.740,40.874,157.852
C07023=1046.139,336.264,-116.716,172.745,40.878,157.853
C07024=1046.147,336.511,-116.752,172.749,40.882,157.854
C07025=1046.154,336.758,-116.788,172.753,40.886,157.855
C07026=1046.161,337.005,-116.824,172.759,40.889,157.856
C07027=1046.167,337.253,-116.860,172.763,40.892,157.857
C07028=1046.175,337.500,-116.896,172.768,40.896,157.858
C07029=1046.181,337.747,-116.932,172.772,40.900,157.859
C07030=1046.189,337.995,-116.968,172.776,40.904,157.860
C07031=1046.196,338.242,-117.004,172.781,40.907,157.862
C07032=1046.203,338.489,-117.041,172.786,40.911,157.863
C07033=1046.210,338.736,-117.077,172.791,40.915,157.864
C07034=1046.218,338.983,-117.113,172.795,40.918,157.865
C07035=1046.225,339.230,-117.149,172.800,40.922,157.866
C07036=1046.232,339.478,-117.186,172.804,40.926,157.867
C07037=1046.240,339.725,-117.222,172.810,40.929,157.868
C07038=1046.247,339.972,-117.258,172.814,40.932,157.869
C07039=1046.254,340.220,-117.295,172.818,40.936,157.870
C07040=1046.261,340.467,-117.331,172.823,40.940,157.871
C07041=1046.268,340.714,-117.367,172.827,40.944,157.872
C07042=1046.275,340.962,-117.404,172.833,40.948,157.874
C07043=1046.283,341.209,-117.440,172.837,40.952,157.875
C07044=1046.290,341.456,-117.476,172.842,40.955,157.876
C07045=1046.297,341.704,-117.512,172.846,40.959,157.877
C07046=1046.305,341.951,-117.549,172.852,40.963,157.878
C07047=1046.311,342.198,-117.586,172.856,40.966,157.879
C07048=1046.319,342.445,-117.622,172.861,40.970,157.880
C07049=1046.326,342.693,-117.659,172.865,40.974,157.881
C07050=1046.333,342.939,-117.695,172.870,40.977,157.882
C07051=1046.340,343.187,-117.732,172.875,40.982,157.884
C07052=1046.348,343.434,-117.768,172.880,40.985,157.885
C07053=1046.355,343.681,-117.806,172.885,40.989,157.886
C07054=1046.362,343.928,-117.842,172.890,40.992,157.887
C07055=1046.369,344.175,-117.879,172.895,40.997,157.888
C07056=1046.376,344.423,-117.916,172.899,41.000,157.889
C07057=1046.384,344.670,-117.952,172.904,41.004,157.890
C07058=1046.391,344.917,-117.990,172.909,41.008,157.892
C07059=1046.398,345.164,-118.026,172.914,41.012,157.893
C07060=1046.406,345.411,-118.063,172.918,41.016,157.894
C07061=1046.412,345.659,-118.100,172.924,41.020,157.895
C07062=1046.420,345.906,-118.137,172.929,41.023,157.896
C07063=1046.428,346.153,-118.175,172.933,41.028,157.897
C07064=1046.435,346.400,-118.210,172.938,41.031,157.899
C07065=1046.442,346.647,-118.248,172.943,41.035,157.900
C07066=1046.449,346.894,-118.285,172.948,41.039,157.901
C07067=1046.458,347.206,-118.331,172.954,41.044,157.902
C07068=1046.468,347.518,-118.378,172.960,41.049,157.904
C07069=1046.477,347.829,-118.425,172.967,41.054,157.905
C07070=1046.486,348.140,-118.472,172.973,41.059,157.907
C07071=1046.493,348.387,-118.509,172.978,41.063,157.908
C07072=1046.501,348.634,-118.546,172.982,41.067,157.909
C07073=1046.508,348.882,-118.583,172.988,41.071,157.910
C07074=1046.515,349.129,-118.621,172.993,41.075,157.912
C07075=1046.523,349.376,-118.658,172.997,41.079,157.913
C07076=1046.531,349.623,-118.695,173.003,41.083,157.914
C07077=1046.538,349.870,-118.733,173.008,41.087,157.915
C07078=1046.545,350.117,-118.770,173.013,41.091,157.916
C07079=1046.553,350.364,-118.807,173.018,41.095,157.918
C07080=1046.560,350.611,-118.845,173.023,41.099,157.919
C07081=1046.568,350.858,-118.882,173.029,41.103,157.920
C07082=1046.575,351.105,-118.920,173.033,41.107,157.921
C07083=1046.582,351.352,-118.957,173.038,41.111,157.922
C07084=1046.589,351.599,-118.995,173.044,41.115,157.924
C07085=1046.597,351.847,-119.032,173.048,41.119,157.925
C07086=1046.604,352.094,-119.070,173.054,41.124,157.926
C07087=1046.611,352.341,-119.107,173.059,41.128,157.928
C07088=1046.619,352.587,-119.146,173.063,41.132,157.929
C07089=1046.626,352.835,-119.183,173.069,41.136,157.930
C07090=1046.634,353.082,-119.221,173.074,41.140,157.931
C07091=1046.641,353.329,-119.259,173.080,41.144,157.933
C07092=1046.649,353.576,-119.297,173.084,41.148,157.934
C07093=1046.657,353.823,-119.334,173.089,41.152,157.935
C07094=1046.664,354.070,-119.371,173.095,41.156,157.936
C07095=1046.671,354.316,-119.409,173.100,41.161,157.938
C07096=1046.679,354.564,-119.447,173.106,41.165,157.939
C07097=1046.686,354.811,-119.485,173.110,41.170,157.940
C07098=1046.694,355.058,-119.523,173.116,41.174,157.941
C07099=1046.701,355.305,-119.561,173.121,41.178,157.943
C07100=1046.709,355.552,-119.599,173.126,41.182,157.944
C07101=1046.716,355.799,-119.636,173.132,41.186,157.945
C07102=1046.724,356.046,-119.675,173.136,41.190,157.947
C07103=1046.731,356.293,-119.713,173.142,41.195,157.948
C07104=1046.739,356.540,-119.751,173.147,41.199,157.949
C07105=1046.746,356.787,-119.788,173.153,41.203,157.951
C07106=1046.754,357.034,-119.827,173.158,41.208,157.952
C07107=1046.762,357.281,-119.864,173.164,41.212,157.953
C07108=1046.768,357.528,-119.903,173.168,41.216,157.954
C07109=1046.776,357.774,-119.942,173.174,41.221,157.956
C07110=1046.784,358.022,-119.979,173.179,41.225,157.957
C07111=1046.791,358.269,-120.018,173.185,41.229,157.958
C07112=1046.799,358.515,-120.056,173.190,41.234,157.960
C07113=1046.807,358.763,-120.095,173.196,41.238,157.961
C07114=1046.814,359.010,-120.133,173.201,41.242,157.962
C07115=1046.821,359.256,-120.171,173.206,41.247,157.964
C07116=1046.829,359.504,-120.210,173.211,41.251,157.965
C07117=1046.837,359.750,-120.248,173.217,41.256,157.966
C07118=1046.844,359.997,-120.286,173.222,41.260,157.968
C07119=1046.852,360.244,-120.325,173.228,41.264,157.969
C07120=1046.859,360.491,-120.363,173.233,41.268,157.970
C07121=1046.867,360.738,-120.402,173.239,41.273,157.972
C07122=1046.875,360.984,-120.440,173.244,41.277,157.973
C07123=1046.884,361.302,-120.490,173.251,41.283,157.975
C07124=1046.894,361.618,-120.539,173.258,41.289,157.977
C07125=1046.904,361.936,-120.588,173.265,41.294,157.978
C07126=1046.914,362.253,-120.639,173.273,41.301,157.980
C07127=1046.921,362.500,-120.677,173.278,41.305,157.982
C07128=1046.930,362.747,-120.716,173.284,41.310,157.983
C07129=1046.937,362.993,-120.755,173.289,41.314,157.984
C07130=1046.945,363.240,-120.794,173.295,41.319,157.986
C07131=1046.952,363.487,-120.833,173.300,41.323,157.987
C07132=1046.960,363.734,-120.871,173.306,41.328,157.989
C07133=1046.967,363.980,-120.911,173.312,41.332,157.990
C07134=1046.975,364.228,-120.950,173.317,41.337,157.991
C07135=1046.982,364.474,-120.989,173.323,41.342,157.993
C07136=1046.990,364.721,-121.028,173.329,41.346,157.994
C07137=1046.997,364.968,-121.067,173.334,41.351,157.996
C07138=1047.006,365.215,-121.106,173.340,41.356,157.997
C07139=1047.013,365.462,-121.145,173.346,41.360,157.999
C07140=1047.021,365.708,-121.184,173.351,41.365,158.000
C07141=1047.028,365.955,-121.223,173.357,41.370,158.002
C07142=1047.036,366.201,-121.262,173.363,41.374,158.003
C07143=1047.044,366.449,-121.301,173.368,41.379,158.004
C07144=1047.051,366.696,-121.341,173.374,41.384,158.006
C07145=1047.059,366.942,-121.380,173.381,41.388,158.007
C07146=1047.067,367.189,-121.419,173.386,41.393,158.009
C07147=1047.075,367.436,-121.459,173.392,41.398,158.010
C07148=1047.082,367.682,-121.498,173.398,41.403,158.012
C07149=1047.090,367.929,-121.537,173.403,41.407,158.013
C07150=1047.098,368.176,-121.577,173.409,41.412,158.015
C07151=1047.106,368.423,-121.616,173.415,41.417,158.016
C07152=1047.114,368.669,-121.656,173.420,41.422,158.018
C07153=1047.121,368.916,-121.696,173.426,41.427,158.019
C07154=1047.129,369.163,-121.734,173.433,41.432,158.021
C07155=1047.137,369.410,-121.774,173.439,41.436,158.022
C07156=1047.146,369.657,-121.813,173.444,41.441,158.024
C07157=1047.153,369.903,-121.853,173.450,41.446,158.025
C07158=1047.161,370.149,-121.892,173.456,41.451,158.027
C07159=1047.169,370.396,-121.932,173.463,41.455,158.028
C07160=1047.177,370.643,-121.972,173.468,41.461,158.030
C07161=1047.185,370.890,-122.012,173.474,41.465,158.031
C07162=1047.193,371.137,-122.051,173.480,41.470,158.033
C07163=1047.200,371.383,-122.091,173.486,41.475,158.034
C07164=1047.208,371.629,-122.130,173.492,41.480,158.036
C07165=1047.216,371.876,-122.170,173.498,41.485,158.037
C07166=1047.224,372.123,-122.211,173.504,41.490,158.039
C07167=1047.232,372.370,-122.251,173.510,41.495,158.041
C07168=1047.240,372.616,-122.291,173.516,41.500,158.042
C07169=1047.247,372.863,-122.331,173.523,41.506,158.044
C07170=1047.255,373.110,-122.371,173.528,41.511,158.045
C07171=1047.263,373.357,-122.411,173.534,41.515,158.047
C07172=1047.270,373.602,-122.451,173.540,41.521,158.048
C07173=1047.278,373.849,-122.491,173.547,41.526,158.050
C07174=1047.287,374.096,-122.531,173.553,41.531,158.052
C07175=1047.295,374.342,-122.571,173.559,41.536,158.053
C07176=1047.302,374.589,-122.611,173.565,41.541,158.055
C07177=1047.310,374.835,-122.652,173.571,41.546,158.056
C07178=1047.318,375.082,-122.692,173.577,41.551,158.058
C07179=1047.329,375.418,-122.747,173.586,41.558,158.060
C07180=1047.340,375.754,-122.802,173.594,41.565,158.062
C07181=1047.351,376.092,-122.857,173.603,41.572,158.065
C07182=1047.363,376.427,-122.912,173.611,41.579,158.067
C07183=1047.371,376.674,-122.953,173.617,41.585,158.069
C07184=1047.378,376.921,-122.993,173.624,41.590,158.070
C07185=1047.386,377.167,-123.033,173.630,41.595,158.072
C07186=1047.394,377.413,-123.074,173.636,41.600,158.073
C07187=1047.402,377.659,-123.115,173.643,41.605,158.075
C07188=1047.411,377.906,-123.156,173.649,41.611,158.077
C07189=1047.419,378.153,-123.195,173.656,41.616,158.079
C07190=1047.427,378.400,-123.236,173.662,41.621,158.080
C07191=1047.435,378.646,-123.277,173.668,41.626,158.082
C07192=1047.443,378.892,-123.317,173.675,41.632,158.084
C07193=1047.451,379.139,-123.358,173.681,41.637,158.085
C07194=1047.459,379.385,-123.399,173.688,41.643,158.087
C07195=1047.467,379.632,-123.440,173.694,41.648,158.089
C07196=1047.475,379.878,-123.480,173.701,41.653,158.090
C07197=1047.483,380.125,-123.522,173.707,41.659,158.092
C07198=1047.491,380.372,-123.563,173.714,41.664,158.094
C07199=1047.500,380.617,-123.604,173.720,41.670,158.096
C07200=1047.508,380.864,-123.644,173.727,41.675,158.097
C07201=1047.516,381.111,-123.686,173.733,41.681,158.099
C07202=1047.524,381.357,-123.727,173.740,41.686,158.101
C07203=1047.532,381.603,-123.768,173.746,41.691,158.102
C07204=1047.541,381.850,-123.809,173.753,41.697,158.104
C07205=1047.548,382.096,-123.850,173.759,41.703,158.106
C07206=1047.556,382.342,-123.892,173.766,41.708,158.108
C07207=1047.565,382.589,-123.933,173.772,41.714,158.110
C07208=1047.572,382.835,-123.975,173.779,41.720,158.111
C07209=1047.581,383.082,-124.016,173.786,41.725,158.113
C07210=1047.589,383.328,-124.057,173.792,41.730,158.115
C07211=1047.597,383.574,-124.098,173.799,41.736,158.117
C07212=1047.606,383.821,-124.140,173.806,41.742,158.118
C07213=1047.614,384.067,-124.181,173.813,41.747,158.120
C07214=1047.622,384.314,-124.223,173.819,41.753,158.122
C07215=1047.630,384.559,-124.264,173.826,41.759,158.124
C07216=1047.639,384.806,-124.305,173.832,41.765,158.126
C07217=1047.646,385.052,-124.347,173.839,41.770,158.127
C07218=1047.655,385.299,-124.389,173.847,41.776,158.129
C07219=1047.664,385.546,-124.430,173.853,41.781,158.131
C07220=1047.672,385.792,-124.472,173.860,41.787,158.133
C07221=1047.681,386.038,-124.514,173.867,41.793,158.135
C07222=1047.689,386.284,-124.555,173.873,41.799,158.137
C07223=1047.697,386.530,-124.597,173.880,41.804,158.138
C07224=1047.706,386.777,-124.639,173.888,41.810,158.140
C07225=1047.714,387.023,-124.680,173.895,41.816,158.142
C07226=1047.722,387.270,-124.722,173.901,41.822,158.144
